// TIA Portal V19 export
FUNCTION_BLOCK "A0302_PareggiatoreTesta_FB"   // FB86, LAD
// stored: MemoryReserve 100, SetENOAutomatically false
   VAR_INPUT
      AreaInterface : "AreaInterface";
      ZSI : "udt_ZoneSafetyInterface";
      DSI_Feed : "udt_DeviceSafetyInterface";
      DSI_Valve : "udt_DeviceSafetyInterface";
      Drive : "TAx_DriveInterface";
      DataIn : Struct
         OP_MoveToPos : Bool;
         Sollevamento : Struct
            OP : "OP_PB";
         END_STRUCT;
         Centraggio : Struct
            OP : "OP_PB";
            AnalSens : Int;
         END_STRUCT;
         Sens { ExternalWritable := 'False'} : Struct
            FTC1_Rall : Bool;   // 2010BF2 - I50.3
            FTC2_Prox_Ls : Bool;   // 2010BF3 - I50.4
            PresenzaMat : Bool;   // FC presenza materiale agganciato lato paregg testa
            FC_Aticoll_Spalla : Bool;
         END_STRUCT;
      END_STRUCT;
      CIn : Struct
         Manager : Struct
            EnableStopDoorOpeningReq { ExternalAccessible := 'False'; ExternalVisible := 'False'; ExternalWritable := 'False'} : Bool;
            EnableStopInPhase { ExternalAccessible := 'False'; ExternalVisible := 'False'; ExternalWritable := 'False'} : Bool;
            EnableStopProgrammed { ExternalAccessible := 'False'; ExternalVisible := 'False'; ExternalWritable := 'False'} : Bool;
            Control_ON { ExternalAccessible := 'False'; ExternalVisible := 'False'; ExternalWritable := 'False'} : Bool;
            MoveToPos { ExternalAccessible := 'False'; ExternalVisible := 'False'; ExternalWritable := 'False'} : Bool;
            Pos { ExternalAccessible := 'False'; ExternalVisible := 'False'; ExternalWritable := 'False'} : LReal;
            Speed : LReal;
            Bloccaggio { ExternalAccessible := 'False'; ExternalVisible := 'False'; ExternalWritable := 'False'} : Struct
               Rest : Bool;
               Work : Bool;
            END_STRUCT;
            Sollevatore { ExternalAccessible := 'False'; ExternalVisible := 'False'; ExternalWritable := 'False'} : Struct
               Rest : Bool;
               Work : Bool;
            END_STRUCT;
            Centraggio { ExternalAccessible := 'False'; ExternalVisible := 'False'; ExternalWritable := 'False'} : Struct
               Rest : Bool;
               Work : Bool;
            END_STRUCT;
         END_STRUCT;
         SemiAut_Pb { ExternalWritable := 'False'} : Bool;
         Bordatrice : Struct
            Ax : "Positioning_EPOS_Machine_COut";
            Sts : Struct
               PosTargetEnable : Bool;
               PosTarget_Reached : Bool;
               In_W_Pos : Bool;
               AtRest : Bool;
            END_STRUCT;
            RegSpalla : Struct
               Infeed_ReqON : Bool;
            END_STRUCT;
         END_STRUCT;
         Rulliera { ExternalWritable := 'False'} : Struct
            Ax_1 : "SpeedMachine_COut";
            Ax_2 : "SpeedMachine_COut";
            Centratori : "ValveMachine_COut";
            Coda : Struct
               Sens : Struct
                  FTC_Rall : Bool;   // Sensori presenza materiale banco rallentamento ingresso
                  FTC_Prox_Ing : Bool;   // Sensori presenza materiale banco limite ingresso
               END_STRUCT;
            END_STRUCT;
            Centro : Struct
               Sens : Struct
                  FTC_Centrale : Bool;   // 2010BF1 - I50.2
               END_STRUCT;
            END_STRUCT;
         END_STRUCT;
         CarroPareggCoda { ExternalWritable := 'False'} : Struct
            Sens : Struct
               FTC_Ingombro_In : Bool;   // 2012BF1 - I50.0
               FTC_Ingombro_Out : Bool;   // 2012BF2 - I50.1
               PresenzaMat : Bool;   // FC presenza materiale agganciato lato paregg coda
            END_STRUCT;
            OilInTargetPressure : Bool;
         END_STRUCT;
         CarriPareggiatori : Struct
            ZoneA0302Entry_Empty { ExternalWritable := 'False'} : Bool;
            ZoneA0302Exit_Empty { ExternalWritable := 'False'} : Bool;
            RequestNewPosition : Bool;
         END_STRUCT;
         Spalle : Struct
            Coda : Struct
               ActualPos : LReal;
            END_STRUCT;
            Testa : Struct
               ActualPos : LReal;
            END_STRUCT;
         END_STRUCT;
         Manipolatore : Struct
            Sollevatore : "ValveMachine_COut";
         END_STRUCT;
         Centratori : Struct
            Sollevamento : "ValveMachine_COut";
         END_STRUCT;
      END_STRUCT;
      Config : Struct
         Ax : "Positioning_DOL_Machine_Config";
         Bloccaggio : "ValveMachine_Config";
         Sollevamento : "ValveMachine_Config";
         Centraggio : "ValveMachine_Config";
         MinDistanzaConSpalla : LReal;
         DelayMissingCondition : Time;
      END_STRUCT;
      HWID : Struct
         Ax_TEL1 : HW_SUBMODULE;
         Enc_IO : HW_SUBMODULE;
      END_STRUCT;
   END_VAR
   VAR_OUTPUT
      MachineInterface : "MachineInterface";
      COut : Struct
         Ax : "Positioning_DOL_Machine_COut";
         Bloccaggio : "ValveMachine_COut";
         Centraggio : "ValveMachine_COut";
         Sollevatore : "ValveMachine_COut";
         Ax_InWPos : Bool;
         Anticipi { ExternalAccessible := 'False'; ExternalVisible := 'False'; ExternalWritable := 'False'} : Struct
            Work : Struct
               Sollevatore : Bool;
               Centraggio : Bool;
            END_STRUCT;
            Rest : Struct
               Sollevatore : Bool;
               Centraggio : Bool;
            END_STRUCT;
         END_STRUCT;
      END_STRUCT;
   END_VAR
   VAR_IN_OUT
      Par : Struct
         Ax : "Positioning_DOL_Machine_Par";
         Ax_Pers : "Positioning_DOL_Machine_Pers_Data";
         Enc : "PosFbk_RTN";
         Ax_Aut : "A0301_Mach_Speed_Par";
         Bloccaggio_Sens : Struct
            "2111B1" : "Analogic_SensorManagement_Par";
            SogliaWork : Real;
         END_STRUCT;
         CarroPareggTesta : Struct
            Delay_StartMove : Time;
            Preset : LReal;
         END_STRUCT;
         Cremaliera : Struct
            Modulo : LReal;
            Passo : LReal;
         END_STRUCT;
      END_STRUCT;
      IEC_SP : Struct
         FTC_Rall : Struct
            TON_PT : Time;
            TOF_PT : Time;
         END_STRUCT;
         FTC_ProxLs : Struct
            TON_PT : Time;
            TOF_PT : Time;
         END_STRUCT;
         FTC_PresentMat : Struct
            TON_PT : Time;
            TOF_PT : Time;
         END_STRUCT;
         Check_2111B1 : Struct
            TON_PT : Time;
         END_STRUCT;
      END_STRUCT;
   END_VAR
   VAR
      Alarm : Struct
         Ax : "Positioning_DOL_Machine_Alr";
         Enc : "PosFbk_Encoder_Alr";
         Bloccaggio : "ValveAlr";
         Centraggio { S7_SetPoint := 'True'} : "ValveAlr";
         Sollevamento { S7_SetPoint := 'True'} : "ValveAlr";
         SensFC_Aticoll_Spalla : Bool;
         Bloccaggio_AnalSens_Issue : Bool;   // Errore soglia lettura pressione su bloccaggio cremaliera
      END_STRUCT;
      Warning : Struct
         Ax : "Positioning_DOL_Machine_Wng";
         Bloccaggio : "ValveMachine_Wng";
         Centraggio { S7_SetPoint := 'True'} : "ValveMachine_Wng";
         Sollevamento { S7_SetPoint := 'True'} : "ValveMachine_Wng";
         MissingCnd : Struct
            OP_REST_Sollevamento : Bool;   // Mancanza comando arresto
            OP_WORK_Sollevamento : Bool;   // Mancanza consenso lavoro
            OP_REST_Centraggio : Bool;   // Mancanza comando arresto
            OP_WORK_Centraggio : Bool;   // Mancanza consenso lavoro
            OP_REST_Bloccaggio : Bool;   // Mancanza comando arresto
            OP_WORK_Bloccaggio : Bool;   // Mancanza consenso lavoro
         END_STRUCT;
         SW_Limit_AntiCollision : Bool;
      END_STRUCT;
      HMI : Struct
         Ax : Struct
            PbPreset : Bool;
            B_Preset_UM2 : Bool;
            PresetValue : LReal;
         END_STRUCT;
      END_STRUCT;
      Sts : Struct
         ReadyForMove : Bool;   // Pronto al movimento
         OP_PTesta_CanMoveFreely : Bool;
         OP_Ax_CanMoveFreely : Bool;
         Op_MoveToPos_Cnd : Bool;
         Sollevamento : Struct
            OP_Rest_Cnd : Bool;
            Op_Work_Cnd : Bool;
         END_STRUCT;
         Centraggio : Struct
            OP_Rest_Cnd : Bool;
            Op_Work_Cnd : Bool;
         END_STRUCT;
      END_STRUCT;
      Ctrl : Struct
         Sollevamento : Struct
            OP_Rest_Man : Bool;
            OP_Work_Man : Bool;
            OP_Rest_Aut : Bool;
            OP_Work_Aut : Bool;
            OP_Rest : Bool;
            OP_Work : Bool;
         END_STRUCT;
         Centraggio : Struct
            OP_Rest_Aut : Bool;
            OP_Work_Aut : Bool;
            OP_Rest_Man : Bool;
            OP_Work_Man : Bool;
            OP_Rest : Bool;
            OP_Work : Bool;
         END_STRUCT;
         Ax : Struct
            OP_MoveToPos_Man : Bool;
            OP_MoveToPos_Aut : Bool;
            OP_MoveToPos : Bool;
         END_STRUCT;
      END_STRUCT;
      AUX : Struct
         OP_MoveToPos : Bool;
         Sollevamento : Struct
            OP_Rest : Bool;
            OP_Work : Bool;
         END_STRUCT;
         Centraggio : Struct
            OP_Rest : Bool;
            OP_Work : Bool;
         END_STRUCT;
      END_STRUCT;
      Ax : "Positioning_DOL_Machine_FB";
      Enc : "PosFbk_SickAFM60";
      Enc_ITF : "PosFbk_ITF";
      Bloccaggio : "ValveMachine_FB";
      Centraggio : "ValveMachine_FB";
      Sollevamento { S7_SetPoint := 'True'} : "ValveMachine_FB";
      TON_Centraggio : Struct
         OP_REST_MissingCnd { S7_SetPoint := 'True'} : TON_TIME;
         OP_WORK_MissingCnd { S7_SetPoint := 'True'} : TON_TIME;
      END_STRUCT;
      TON_Sollevamento : Struct
         OP_REST_MissingCnd { S7_SetPoint := 'True'} : TON_TIME;
         OP_WORK_MissingCnd { S7_SetPoint := 'True'} : TON_TIME;
      END_STRUCT;
      TON_Bloccaggio : Struct
         OP_REST_MissingCnd { S7_SetPoint := 'True'} : TON_TIME;
         OP_WORK_MissingCnd { S7_SetPoint := 'True'} : TON_TIME;
      END_STRUCT;
      IEC_FTC_Rall : Struct
         TON_Delay : IEC_TIMER;
         TOF_Delay { S7_SetPoint := 'True'} : IEC_TIMER;
         FTC_On { S7_SetPoint := 'True'} : Bool;
      END_STRUCT;
      IEC_FTC_ProxLs : Struct
         TON_Delay : IEC_TIMER;
         TOF_Delay { S7_SetPoint := 'True'} : IEC_TIMER;
         FTC_On { S7_SetPoint := 'True'} : Bool;
      END_STRUCT;
      IEC_FTC_PresentMat : Struct
         TON_Delay : IEC_TIMER;
         TOF_Delay { S7_SetPoint := 'True'} : IEC_TIMER;
         FTC_On { S7_SetPoint := 'True'} : Bool;
      END_STRUCT;
      IEC_DelayCheck_2111B1 : IEC_TIMER;
      Bloccaggio_AnalSens { S7_SetPoint := 'True'} : "AnalogThreshold";
      CarroTesta : Struct
         RimanenzaPos : LReal;
         PassoReq : LReal;
         PosBattutePz : LReal;
         SemiBeamLen : LReal;
         NrPassiReq : LReal;
         Pos { ExternalAccessible := 'False'; ExternalVisible := 'False'; ExternalWritable := 'False'} : LReal;   // Posizione calcolata in funzione della cremaliera
      END_STRUCT;
      TON_DistanzaOK : IEC_TIMER;
      TON_Anticipi : Struct
         Rest : Struct
            Sollevamento { S7_SetPoint := 'True'} : IEC_TIMER;
            Centraggio : IEC_TIMER;
         END_STRUCT;
         Work : Struct
            Sollevamento : IEC_TIMER;
            Centraggio { S7_SetPoint := 'True'} : IEC_TIMER;
         END_STRUCT;
      END_STRUCT;
   END_VAR
   VAR_TEMP
      PE : Struct
         OP_MoveToPos : Bool;
         Sollevamento : Struct
            OP_Rest : Bool;
            OP_Work : Bool;
         END_STRUCT;
         Centraggio : Struct
            OP_Rest : Bool;
            OP_Work : Bool;
         END_STRUCT;
      END_STRUCT;
      ActualDifference : LReal;
   END_VAR
   VAR CONSTANT
      RACK_STEP : LReal;   // Passo Cremagliera mm
   END_VAR
   VAR_TEMP   // added for the SCL form of the ladder/FBD networks
      _w1 : Bool;
      _w2 : Bool;
      _w3 : Bool;
      _w4 : Bool;
      _w5 : Bool;
      _w6 : Bool;
      _w7 : Bool;
      _w8 : Bool;
      _w9 : Bool;
      _w10 : Bool;
      _w11 : Bool;
      _w12 : Bool;
   END_VAR
BEGIN

REGION Network 1 (SCL): Reset allarmi
   IF #AreaInterface.RstAlarms THEN
       #Alarm.SensFC_Aticoll_Spalla := FALSE;
       #Alarm.Bloccaggio_AnalSens_Issue := FALSE;
   END_IF;
END_REGION

REGION Network 2: <+>
END_REGION

REGION Network 3: Anticipi Movimento LAVORO
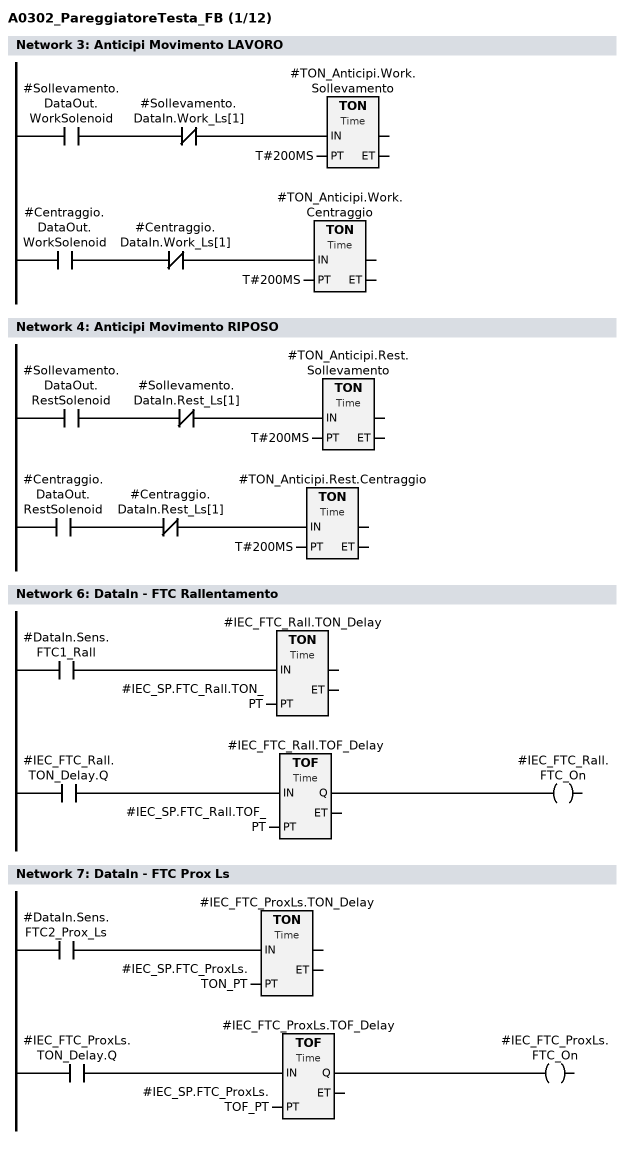
   RUNG wire#powerrail
      Contact( #Sollevamento.DataOut.WorkSolenoid )
      I_Contact( #Sollevamento.DataIn.Work_Ls[1] )
      { S7_Templates := "time_type := Time" } #TON_Anticipi.Work.Sollevamento.TON(pt := T#200MS, et =>)
   END_RUNG
   RUNG wire#powerrail
      Contact( #Centraggio.DataOut.WorkSolenoid )
      I_Contact( #Centraggio.DataIn.Work_Ls[1] )
      { S7_Templates := "time_type := Time" } #TON_Anticipi.Work.Centraggio.TON(pt := T#200MS, et =>)
   END_RUNG
   // the same network as SCL:
   #TON_Anticipi.Work.Sollevamento.TON(IN := #Sollevamento.DataOut.WorkSolenoid AND NOT #Sollevamento.DataIn.Work_Ls[1],
                           PT := T#200MS);
   #TON_Anticipi.Work.Centraggio.TON(IN := #Centraggio.DataOut.WorkSolenoid AND NOT #Centraggio.DataIn.Work_Ls[1],
                           PT := T#200MS);
END_REGION

REGION Network 4: Anticipi Movimento RIPOSO
   RUNG wire#powerrail
      Contact( #Sollevamento.DataOut.RestSolenoid )
      I_Contact( #Sollevamento.DataIn.Rest_Ls[1] )
      { S7_Templates := "time_type := Time" } #TON_Anticipi.Rest.Sollevamento.TON(pt := T#200MS, et =>)
   END_RUNG
   RUNG wire#powerrail
      Contact( #Centraggio.DataOut.RestSolenoid )
      I_Contact( #Centraggio.DataIn.Rest_Ls[1] )
      { S7_Templates := "time_type := Time" } #TON_Anticipi.Rest.Centraggio.TON(pt := T#200MS, et =>)
   END_RUNG
   // the same network as SCL:
   #TON_Anticipi.Rest.Sollevamento.TON(IN := #Sollevamento.DataOut.RestSolenoid AND NOT #Sollevamento.DataIn.Rest_Ls[1],
                           PT := T#200MS);
   #TON_Anticipi.Rest.Centraggio.TON(IN := #Centraggio.DataOut.RestSolenoid AND NOT #Centraggio.DataIn.Rest_Ls[1],
                           PT := T#200MS);
END_REGION

REGION Network 5: <+>
END_REGION

REGION Network 6: DataIn - FTC Rallentamento
   RUNG wire#powerrail
      Contact( #DataIn.Sens.FTC1_Rall )
      { S7_Templates := "time_type := Time" } #IEC_FTC_Rall.TON_Delay.TON(pt := #IEC_SP.FTC_Rall.TON_PT, et =>)
   END_RUNG
   RUNG wire#powerrail
      Contact( #IEC_FTC_Rall.TON_Delay.Q )
      { S7_Templates := "time_type := Time" } #IEC_FTC_Rall.TOF_Delay.TOF(pt := #IEC_SP.FTC_Rall.TOF_PT, et =>)
      Coil( #IEC_FTC_Rall.FTC_On )
   END_RUNG
   // the same network as SCL:
   #IEC_FTC_Rall.TON_Delay.TON(IN := #DataIn.Sens.FTC1_Rall, PT := #IEC_SP.FTC_Rall.TON_PT);
   #IEC_FTC_Rall.TOF_Delay.TOF(IN := #IEC_FTC_Rall.TON_Delay.Q, PT := #IEC_SP.FTC_Rall.TOF_PT);
   #IEC_FTC_Rall.FTC_On := #IEC_FTC_Rall.TOF_Delay.Q;
END_REGION

REGION Network 7: DataIn - FTC Prox Ls
   RUNG wire#powerrail
      Contact( #DataIn.Sens.FTC2_Prox_Ls )
      { S7_Templates := "time_type := Time" } #IEC_FTC_ProxLs.TON_Delay.TON(pt := #IEC_SP.FTC_ProxLs.TON_PT, et =>)
   END_RUNG
   RUNG wire#powerrail
      Contact( #IEC_FTC_ProxLs.TON_Delay.Q )
      { S7_Templates := "time_type := Time" } #IEC_FTC_ProxLs.TOF_Delay.TOF(pt := #IEC_SP.FTC_ProxLs.TOF_PT, et =>)
      Coil( #IEC_FTC_ProxLs.FTC_On )
   END_RUNG
   // the same network as SCL:
   #IEC_FTC_ProxLs.TON_Delay.TON(IN := #DataIn.Sens.FTC2_Prox_Ls, PT := #IEC_SP.FTC_ProxLs.TON_PT);
   #IEC_FTC_ProxLs.TOF_Delay.TOF(IN := #IEC_FTC_ProxLs.TON_Delay.Q, PT := #IEC_SP.FTC_ProxLs.TOF_PT);
   #IEC_FTC_ProxLs.FTC_On := #IEC_FTC_ProxLs.TOF_Delay.Q;
END_REGION

REGION Network 8: DataIn - FTC Presenza materiale
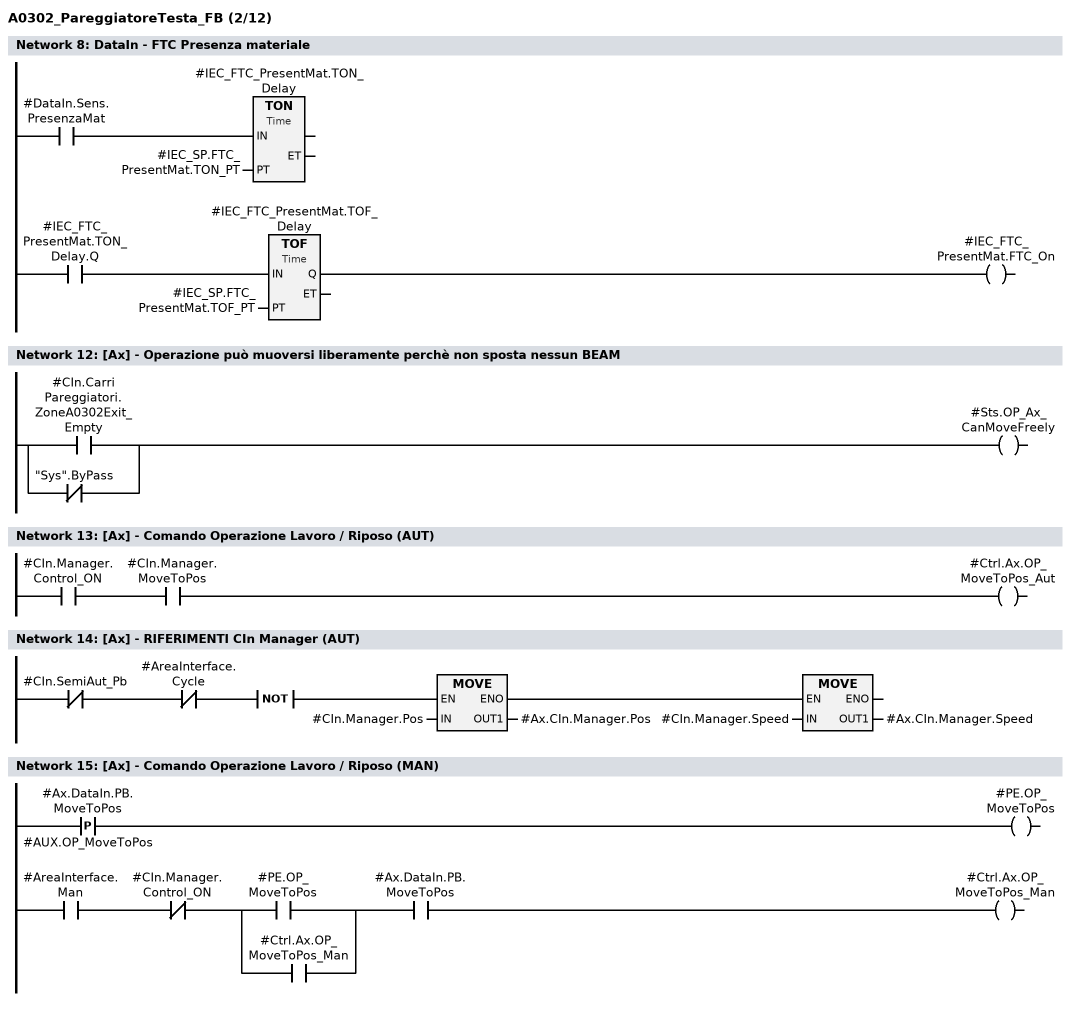
   RUNG wire#powerrail
      Contact( #DataIn.Sens.PresenzaMat )
      { S7_Templates := "time_type := Time" } #IEC_FTC_PresentMat.TON_Delay.TON(pt := #IEC_SP.FTC_PresentMat.TON_PT, et =>)
   END_RUNG
   RUNG wire#powerrail
      Contact( #IEC_FTC_PresentMat.TON_Delay.Q )
      { S7_Templates := "time_type := Time" } #IEC_FTC_PresentMat.TOF_Delay.TOF(pt := #IEC_SP.FTC_PresentMat.TOF_PT, et =>)
      Coil( #IEC_FTC_PresentMat.FTC_On )
   END_RUNG
   // the same network as SCL:
   #IEC_FTC_PresentMat.TON_Delay.TON(IN := #DataIn.Sens.PresenzaMat, PT := #IEC_SP.FTC_PresentMat.TON_PT);
   #IEC_FTC_PresentMat.TOF_Delay.TOF(IN := #IEC_FTC_PresentMat.TON_Delay.Q, PT := #IEC_SP.FTC_PresentMat.TOF_PT);
   #IEC_FTC_PresentMat.FTC_On := #IEC_FTC_PresentMat.TOF_Delay.Q;
END_REGION

REGION Network 9: <+>
END_REGION

REGION Network 10: <<< CARRO PAREGGIATORE TESTA >>>
END_REGION

REGION Network 11: <+>
END_REGION

REGION Network 12: [Ax] - Operazione può muoversi liberamente perchè non sposta nessun BEAM
   RUNG wire#powerrail
      Contact( #CIn.CarriPareggiatori.ZoneA0302Exit_Empty )
      wire#w1
      Coil( #Sts.OP_Ax_CanMoveFreely )
   END_RUNG
   RUNG wire#powerrail
      I_Contact( "Sys".ByPass )
   END_RUNG wire#w1
   // the same network as SCL:
   #Sts.OP_Ax_CanMoveFreely := #CIn.CarriPareggiatori.ZoneA0302Exit_Empty OR NOT "Sys".ByPass;
END_REGION

REGION Network 13: [Ax] - Comando Operazione Lavoro / Riposo (AUT)
   RUNG wire#powerrail
      Contact( #CIn.Manager.Control_ON )
      Contact( #CIn.Manager.MoveToPos )
      Coil( #Ctrl.Ax.OP_MoveToPos_Aut )
   END_RUNG
   // the same network as SCL:
   #Ctrl.Ax.OP_MoveToPos_Aut := #CIn.Manager.Control_ON AND #CIn.Manager.MoveToPos;
END_REGION

REGION Network 14: [Ax] - RIFERIMENTI CIn Manager (AUT)
   RUNG wire#powerrail
      I_Contact( #CIn.SemiAut_Pb )
      I_Contact( #AreaInterface.Cycle )
      Not()
      Move(in := #CIn.Manager.Pos, out1 => #Ax.CIn.Manager.Pos)
      Move(in := #CIn.Manager.Speed, out1 => #Ax.CIn.Manager.Speed)
   END_RUNG
   // the same network as SCL:
   IF NOT (NOT #CIn.SemiAut_Pb AND NOT #AreaInterface.Cycle) THEN
       #Ax.CIn.Manager.Pos := #CIn.Manager.Pos;
       #Ax.CIn.Manager.Speed := #CIn.Manager.Speed;
   END_IF;
END_REGION

REGION Network 15: [Ax] - Comando Operazione Lavoro / Riposo (MAN)
   RUNG wire#powerrail
      P_Contact(operand := #Ax.DataIn.PB.MoveToPos, bit := #AUX.OP_MoveToPos)
      Coil( #PE.OP_MoveToPos )
   END_RUNG
   RUNG wire#powerrail
      Contact( #AreaInterface.Man )
      I_Contact( #CIn.Manager.Control_ON )
      wire#w1
      Contact( #PE.OP_MoveToPos )
      wire#w2
      Contact( #Ax.DataIn.PB.MoveToPos )
      Coil( #Ctrl.Ax.OP_MoveToPos_Man )
   END_RUNG
   RUNG wire#w1
      Contact( #Ctrl.Ax.OP_MoveToPos_Man )
   END_RUNG wire#w2
   // the same network as SCL:
   #_w1 := #Ax.DataIn.PB.MoveToPos AND NOT #AUX.OP_MoveToPos;   // rising edge of #Ax.DataIn.PB.MoveToPos
   #AUX.OP_MoveToPos := #Ax.DataIn.PB.MoveToPos;
   #PE.OP_MoveToPos := #_w1;
   #Ctrl.Ax.OP_MoveToPos_Man := #AreaInterface.Man AND NOT #CIn.Manager.Control_ON AND (#PE.OP_MoveToPos OR #Ctrl.Ax.OP_MoveToPos_Man) AND #Ax.DataIn.PB.MoveToPos;
END_REGION

REGION Network 16: <+>
END_REGION

REGION Network 17: [Sollevam + Centraggio] - Operazione può muoversi liberamente perchè non sposta nessun BEAM
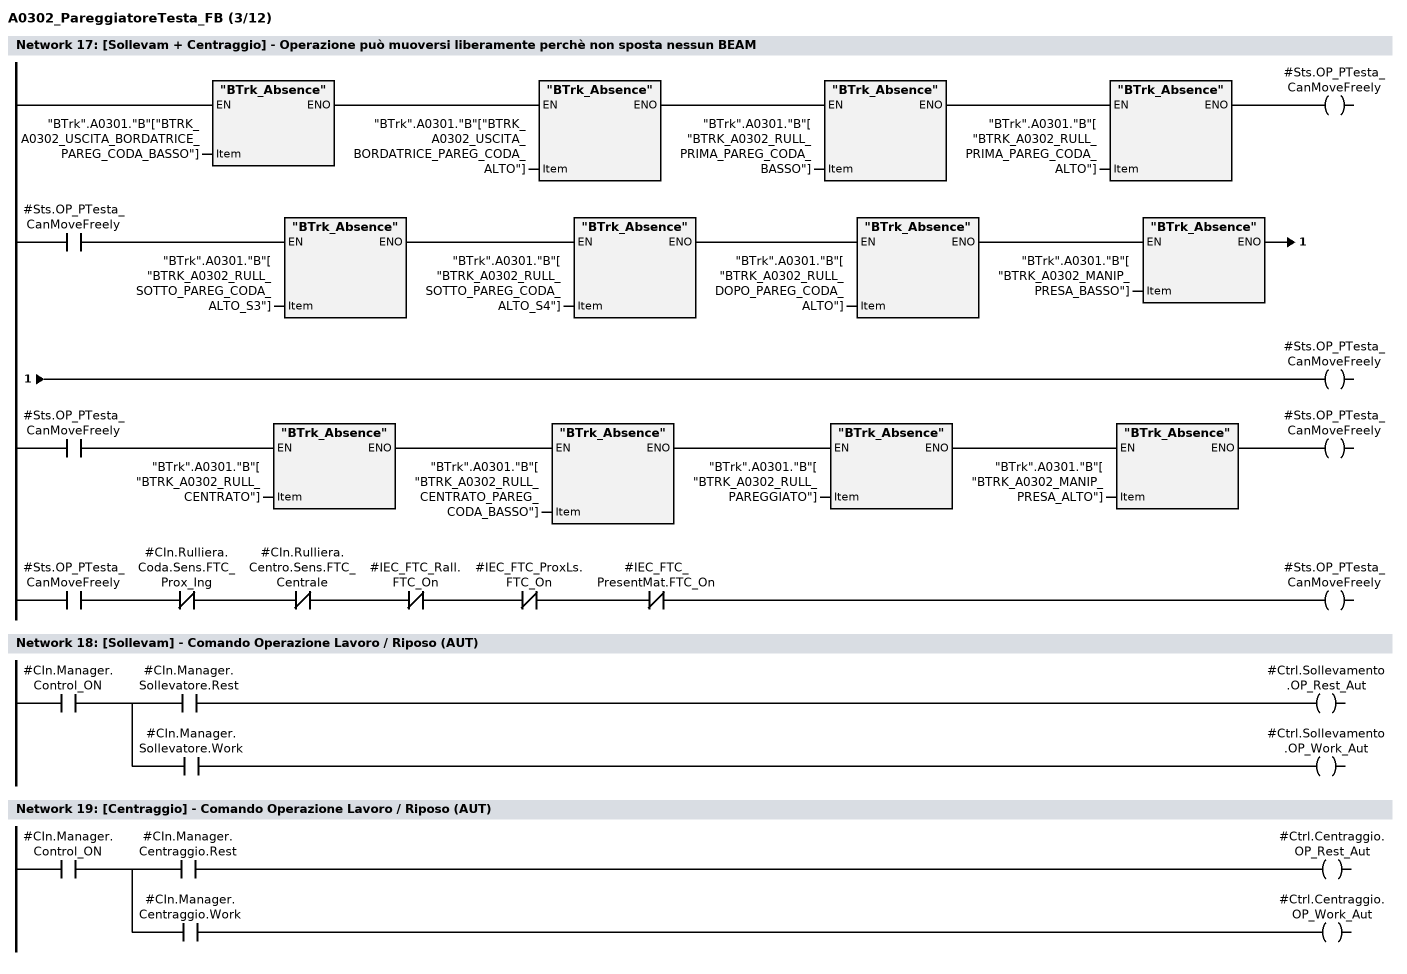
   RUNG wire#powerrail
      "BTrk_Absence"(Item := "BTrk".A0301."B"["BTRK_A0302_USCITA_BORDATRICE_PAREG_CODA_BASSO"])
      "BTrk_Absence"(Item := "BTrk".A0301."B"["BTRK_A0302_USCITA_BORDATRICE_PAREG_CODA_ALTO"])
      "BTrk_Absence"(Item := "BTrk".A0301."B"["BTRK_A0302_RULL_PRIMA_PAREG_CODA_BASSO"])
      "BTrk_Absence"(Item := "BTrk".A0301."B"["BTRK_A0302_RULL_PRIMA_PAREG_CODA_ALTO"])
      Coil( #Sts.OP_PTesta_CanMoveFreely )
   END_RUNG
   RUNG wire#powerrail
      Contact( #Sts.OP_PTesta_CanMoveFreely )
      "BTrk_Absence"(Item := "BTrk".A0301."B"["BTRK_A0302_RULL_SOTTO_PAREG_CODA_ALTO_S3"])
      "BTrk_Absence"(Item := "BTrk".A0301."B"["BTRK_A0302_RULL_SOTTO_PAREG_CODA_ALTO_S4"])
      "BTrk_Absence"(Item := "BTrk".A0301."B"["BTRK_A0302_RULL_DOPO_PAREG_CODA_ALTO"])
      "BTrk_Absence"(Item := "BTrk".A0301."B"["BTRK_A0302_MANIP_PRESA_BASSO"])
      Coil( #Sts.OP_PTesta_CanMoveFreely )
   END_RUNG
   RUNG wire#powerrail
      Contact( #Sts.OP_PTesta_CanMoveFreely )
      "BTrk_Absence"(Item := "BTrk".A0301."B"["BTRK_A0302_RULL_CENTRATO"])
      "BTrk_Absence"(Item := "BTrk".A0301."B"["BTRK_A0302_RULL_CENTRATO_PAREG_CODA_BASSO"])
      "BTrk_Absence"(Item := "BTrk".A0301."B"["BTRK_A0302_RULL_PAREGGIATO"])
      "BTrk_Absence"(Item := "BTrk".A0301."B"["BTRK_A0302_MANIP_PRESA_ALTO"])
      Coil( #Sts.OP_PTesta_CanMoveFreely )
   END_RUNG
   RUNG wire#powerrail
      Contact( #Sts.OP_PTesta_CanMoveFreely )
      I_Contact( #CIn.Rulliera.Coda.Sens.FTC_Prox_Ing )
      I_Contact( #CIn.Rulliera.Centro.Sens.FTC_Centrale )
      I_Contact( #IEC_FTC_Rall.FTC_On )
      I_Contact( #IEC_FTC_ProxLs.FTC_On )
      I_Contact( #IEC_FTC_PresentMat.FTC_On )
      Coil( #Sts.OP_PTesta_CanMoveFreely )
   END_RUNG
   // the same network as SCL:
   "BTrk_Absence"(Item := "BTrk".A0301."B"["BTRK_A0302_USCITA_BORDATRICE_PAREG_CODA_BASSO"], ENO => #_w1);
   "BTrk_Absence"(EN := #_w1,
                  Item := "BTrk".A0301."B"["BTRK_A0302_USCITA_BORDATRICE_PAREG_CODA_ALTO"],
                  ENO => #_w2);
   "BTrk_Absence"(EN := #_w2, Item := "BTrk".A0301."B"["BTRK_A0302_RULL_PRIMA_PAREG_CODA_BASSO"], ENO => #_w3);
   "BTrk_Absence"(EN := #_w3, Item := "BTrk".A0301."B"["BTRK_A0302_RULL_PRIMA_PAREG_CODA_ALTO"], ENO => #_w4);
   #Sts.OP_PTesta_CanMoveFreely := #_w4;
   "BTrk_Absence"(EN := #Sts.OP_PTesta_CanMoveFreely,
                  Item := "BTrk".A0301."B"["BTRK_A0302_RULL_SOTTO_PAREG_CODA_ALTO_S3"],
                  ENO => #_w5);
   "BTrk_Absence"(EN := #_w5, Item := "BTrk".A0301."B"["BTRK_A0302_RULL_SOTTO_PAREG_CODA_ALTO_S4"], ENO => #_w6);
   "BTrk_Absence"(EN := #_w6, Item := "BTrk".A0301."B"["BTRK_A0302_RULL_DOPO_PAREG_CODA_ALTO"], ENO => #_w7);
   "BTrk_Absence"(EN := #_w7, Item := "BTrk".A0301."B"["BTRK_A0302_MANIP_PRESA_BASSO"], ENO => #_w8);
   #Sts.OP_PTesta_CanMoveFreely := #_w8;
   "BTrk_Absence"(EN := #Sts.OP_PTesta_CanMoveFreely,
                  Item := "BTrk".A0301."B"["BTRK_A0302_RULL_CENTRATO"],
                  ENO => #_w9);
   "BTrk_Absence"(EN := #_w9,
                  Item := "BTrk".A0301."B"["BTRK_A0302_RULL_CENTRATO_PAREG_CODA_BASSO"],
                  ENO => #_w10);
   "BTrk_Absence"(EN := #_w10, Item := "BTrk".A0301."B"["BTRK_A0302_RULL_PAREGGIATO"], ENO => #_w11);
   "BTrk_Absence"(EN := #_w11, Item := "BTrk".A0301."B"["BTRK_A0302_MANIP_PRESA_ALTO"], ENO => #_w12);
   #Sts.OP_PTesta_CanMoveFreely := #_w12;
   #Sts.OP_PTesta_CanMoveFreely := #Sts.OP_PTesta_CanMoveFreely AND NOT #CIn.Rulliera.Coda.Sens.FTC_Prox_Ing AND NOT #CIn.Rulliera.Centro.Sens.FTC_Centrale AND NOT #IEC_FTC_Rall.FTC_On AND NOT #IEC_FTC_ProxLs.FTC_On AND NOT #IEC_FTC_PresentMat.FTC_On;
END_REGION

REGION Network 18: [Sollevam] - Comando Operazione Lavoro / Riposo (AUT)
   RUNG wire#powerrail
      Contact( #CIn.Manager.Control_ON )
      wire#w1
      Contact( #CIn.Manager.Sollevatore.Rest )
      Coil( #Ctrl.Sollevamento.OP_Rest_Aut )
   END_RUNG
   RUNG wire#w1
      Contact( #CIn.Manager.Sollevatore.Work )
      Coil( #Ctrl.Sollevamento.OP_Work_Aut )
   END_RUNG
   // the same network as SCL:
   #Ctrl.Sollevamento.OP_Rest_Aut := #CIn.Manager.Control_ON AND #CIn.Manager.Sollevatore.Rest;
   #Ctrl.Sollevamento.OP_Work_Aut := #CIn.Manager.Control_ON AND #CIn.Manager.Sollevatore.Work;
END_REGION

REGION Network 19: [Centraggio] - Comando Operazione Lavoro / Riposo (AUT)
   RUNG wire#powerrail
      Contact( #CIn.Manager.Control_ON )
      wire#w1
      Contact( #CIn.Manager.Centraggio.Rest )
      Coil( #Ctrl.Centraggio.OP_Rest_Aut )
   END_RUNG
   RUNG wire#w1
      Contact( #CIn.Manager.Centraggio.Work )
      Coil( #Ctrl.Centraggio.OP_Work_Aut )
   END_RUNG
   // the same network as SCL:
   #Ctrl.Centraggio.OP_Rest_Aut := #CIn.Manager.Control_ON AND #CIn.Manager.Centraggio.Rest;
   #Ctrl.Centraggio.OP_Work_Aut := #CIn.Manager.Control_ON AND #CIn.Manager.Centraggio.Work;
END_REGION

REGION Network 20: <+>
END_REGION

REGION Network 21: [Sollevam] - Comando Operazione Lavoro / Riposo (MAN)
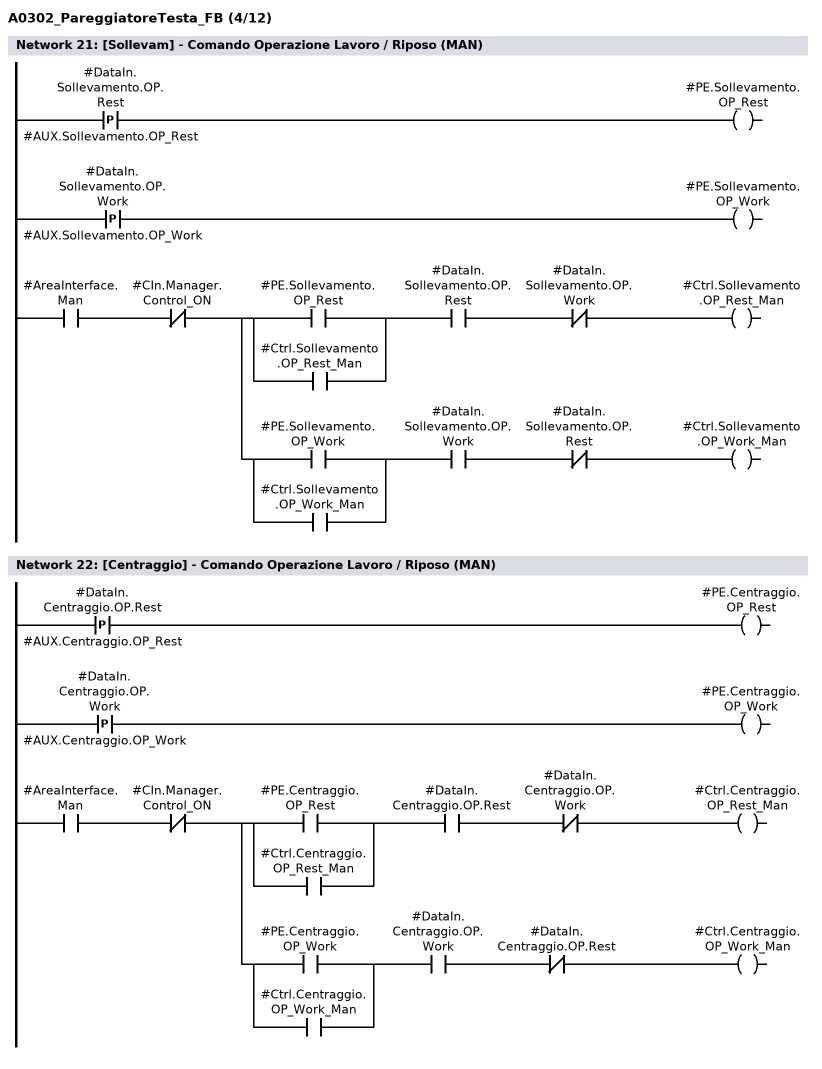
   RUNG wire#powerrail
      P_Contact(operand := #DataIn.Sollevamento.OP.Rest, bit := #AUX.Sollevamento.OP_Rest)
      Coil( #PE.Sollevamento.OP_Rest )
   END_RUNG
   RUNG wire#powerrail
      P_Contact(operand := #DataIn.Sollevamento.OP.Work, bit := #AUX.Sollevamento.OP_Work)
      Coil( #PE.Sollevamento.OP_Work )
   END_RUNG
   RUNG wire#powerrail
      Contact( #AreaInterface.Man )
      I_Contact( #CIn.Manager.Control_ON )
      wire#w1
      Contact( #PE.Sollevamento.OP_Rest )
      wire#w2
      Contact( #DataIn.Sollevamento.OP.Rest )
      I_Contact( #DataIn.Sollevamento.OP.Work )
      Coil( #Ctrl.Sollevamento.OP_Rest_Man )
   END_RUNG
   RUNG wire#w1
      Contact( #Ctrl.Sollevamento.OP_Rest_Man )
   END_RUNG wire#w2
   RUNG wire#w1
      Contact( #PE.Sollevamento.OP_Work )
      wire#w3
      Contact( #DataIn.Sollevamento.OP.Work )
      I_Contact( #DataIn.Sollevamento.OP.Rest )
      Coil( #Ctrl.Sollevamento.OP_Work_Man )
   END_RUNG
   RUNG wire#w1
      Contact( #Ctrl.Sollevamento.OP_Work_Man )
   END_RUNG wire#w3
   // the same network as SCL:
   #_w1 := #DataIn.Sollevamento.OP.Rest AND NOT #AUX.Sollevamento.OP_Rest;   // rising edge of #DataIn.Sollevamento.OP.Rest
   #AUX.Sollevamento.OP_Rest := #DataIn.Sollevamento.OP.Rest;
   #PE.Sollevamento.OP_Rest := #_w1;
   #_w2 := #DataIn.Sollevamento.OP.Work AND NOT #AUX.Sollevamento.OP_Work;   // rising edge of #DataIn.Sollevamento.OP.Work
   #AUX.Sollevamento.OP_Work := #DataIn.Sollevamento.OP.Work;
   #PE.Sollevamento.OP_Work := #_w2;
   #_w3 := #AreaInterface.Man AND NOT #CIn.Manager.Control_ON;
   #Ctrl.Sollevamento.OP_Rest_Man := #_w3 AND (#PE.Sollevamento.OP_Rest OR #Ctrl.Sollevamento.OP_Rest_Man) AND #DataIn.Sollevamento.OP.Rest AND NOT #DataIn.Sollevamento.OP.Work;
   #Ctrl.Sollevamento.OP_Work_Man := #_w3 AND (#PE.Sollevamento.OP_Work OR #Ctrl.Sollevamento.OP_Work_Man) AND #DataIn.Sollevamento.OP.Work AND NOT #DataIn.Sollevamento.OP.Rest;
END_REGION

REGION Network 22: [Centraggio] - Comando Operazione Lavoro / Riposo (MAN)
   RUNG wire#powerrail
      P_Contact(operand := #DataIn.Centraggio.OP.Rest, bit := #AUX.Centraggio.OP_Rest)
      Coil( #PE.Centraggio.OP_Rest )
   END_RUNG
   RUNG wire#powerrail
      P_Contact(operand := #DataIn.Centraggio.OP.Work, bit := #AUX.Centraggio.OP_Work)
      Coil( #PE.Centraggio.OP_Work )
   END_RUNG
   RUNG wire#powerrail
      Contact( #AreaInterface.Man )
      I_Contact( #CIn.Manager.Control_ON )
      wire#w1
      Contact( #PE.Centraggio.OP_Rest )
      wire#w2
      Contact( #DataIn.Centraggio.OP.Rest )
      I_Contact( #DataIn.Centraggio.OP.Work )
      Coil( #Ctrl.Centraggio.OP_Rest_Man )
   END_RUNG
   RUNG wire#w1
      Contact( #Ctrl.Centraggio.OP_Rest_Man )
   END_RUNG wire#w2
   RUNG wire#w1
      Contact( #PE.Centraggio.OP_Work )
      wire#w3
      Contact( #DataIn.Centraggio.OP.Work )
      I_Contact( #DataIn.Centraggio.OP.Rest )
      Coil( #Ctrl.Centraggio.OP_Work_Man )
   END_RUNG
   RUNG wire#w1
      Contact( #Ctrl.Centraggio.OP_Work_Man )
   END_RUNG wire#w3
   // the same network as SCL:
   #_w1 := #DataIn.Centraggio.OP.Rest AND NOT #AUX.Centraggio.OP_Rest;   // rising edge of #DataIn.Centraggio.OP.Rest
   #AUX.Centraggio.OP_Rest := #DataIn.Centraggio.OP.Rest;
   #PE.Centraggio.OP_Rest := #_w1;
   #_w2 := #DataIn.Centraggio.OP.Work AND NOT #AUX.Centraggio.OP_Work;   // rising edge of #DataIn.Centraggio.OP.Work
   #AUX.Centraggio.OP_Work := #DataIn.Centraggio.OP.Work;
   #PE.Centraggio.OP_Work := #_w2;
   #_w3 := #AreaInterface.Man AND NOT #CIn.Manager.Control_ON;
   #Ctrl.Centraggio.OP_Rest_Man := #_w3 AND (#PE.Centraggio.OP_Rest OR #Ctrl.Centraggio.OP_Rest_Man) AND #DataIn.Centraggio.OP.Rest AND NOT #DataIn.Centraggio.OP.Work;
   #Ctrl.Centraggio.OP_Work_Man := #_w3 AND (#PE.Centraggio.OP_Work OR #Ctrl.Centraggio.OP_Work_Man) AND #DataIn.Centraggio.OP.Work AND NOT #DataIn.Centraggio.OP.Rest;
END_REGION

REGION Network 23: <+>
END_REGION

REGION Network 24: Carro Pareggiatore di Testa - Cumulativo Operazione Lavoro / Riposo (ALL)
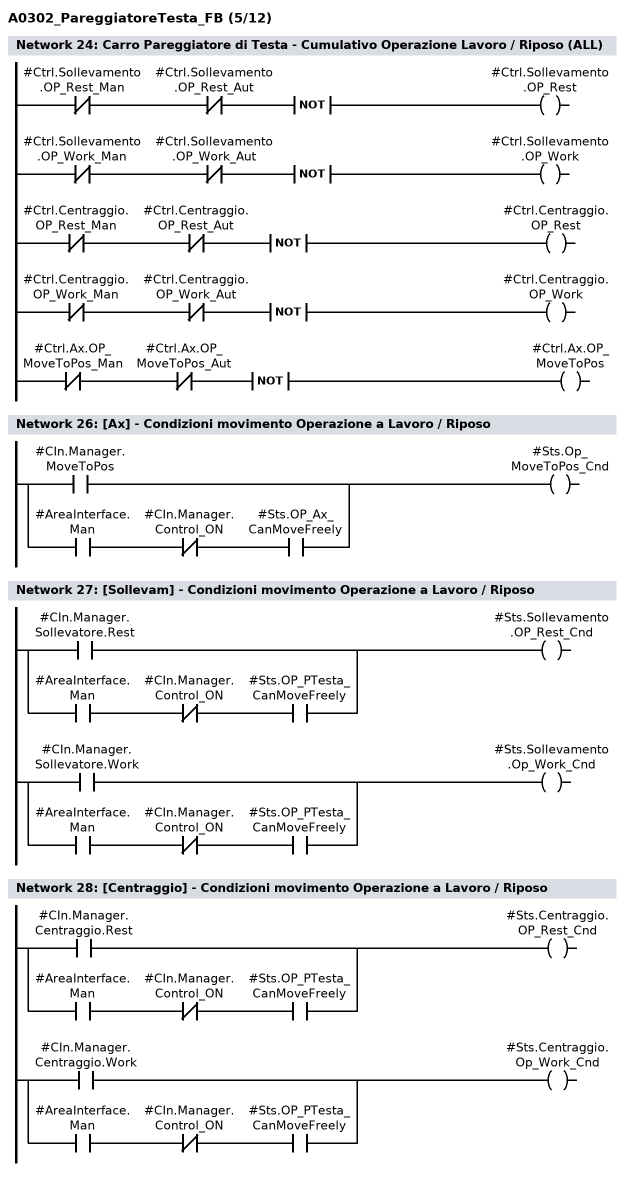
   RUNG wire#powerrail
      I_Contact( #Ctrl.Sollevamento.OP_Rest_Man )
      I_Contact( #Ctrl.Sollevamento.OP_Rest_Aut )
      Not()
      Coil( #Ctrl.Sollevamento.OP_Rest )
   END_RUNG
   RUNG wire#powerrail
      I_Contact( #Ctrl.Sollevamento.OP_Work_Man )
      I_Contact( #Ctrl.Sollevamento.OP_Work_Aut )
      Not()
      Coil( #Ctrl.Sollevamento.OP_Work )
   END_RUNG
   RUNG wire#powerrail
      I_Contact( #Ctrl.Centraggio.OP_Rest_Man )
      I_Contact( #Ctrl.Centraggio.OP_Rest_Aut )
      Not()
      Coil( #Ctrl.Centraggio.OP_Rest )
   END_RUNG
   RUNG wire#powerrail
      I_Contact( #Ctrl.Centraggio.OP_Work_Man )
      I_Contact( #Ctrl.Centraggio.OP_Work_Aut )
      Not()
      Coil( #Ctrl.Centraggio.OP_Work )
   END_RUNG
   RUNG wire#powerrail
      I_Contact( #Ctrl.Ax.OP_MoveToPos_Man )
      I_Contact( #Ctrl.Ax.OP_MoveToPos_Aut )
      Not()
      Coil( #Ctrl.Ax.OP_MoveToPos )
   END_RUNG
   // the same network as SCL:
   #Ctrl.Sollevamento.OP_Rest := NOT (NOT #Ctrl.Sollevamento.OP_Rest_Man AND NOT #Ctrl.Sollevamento.OP_Rest_Aut);
   #Ctrl.Sollevamento.OP_Work := NOT (NOT #Ctrl.Sollevamento.OP_Work_Man AND NOT #Ctrl.Sollevamento.OP_Work_Aut);
   #Ctrl.Centraggio.OP_Rest := NOT (NOT #Ctrl.Centraggio.OP_Rest_Man AND NOT #Ctrl.Centraggio.OP_Rest_Aut);
   #Ctrl.Centraggio.OP_Work := NOT (NOT #Ctrl.Centraggio.OP_Work_Man AND NOT #Ctrl.Centraggio.OP_Work_Aut);
   #Ctrl.Ax.OP_MoveToPos := NOT (NOT #Ctrl.Ax.OP_MoveToPos_Man AND NOT #Ctrl.Ax.OP_MoveToPos_Aut);
END_REGION

REGION Network 25: <+>
END_REGION

REGION Network 26: [Ax] - Condizioni movimento Operazione a Lavoro / Riposo
   RUNG wire#powerrail
      Contact( #CIn.Manager.MoveToPos )
      wire#w1
      Coil( #Sts.Op_MoveToPos_Cnd )
   END_RUNG
   RUNG wire#powerrail
      Contact( #AreaInterface.Man )
      I_Contact( #CIn.Manager.Control_ON )
      Contact( #Sts.OP_Ax_CanMoveFreely )
   END_RUNG wire#w1
   // the same network as SCL:
   #Sts.Op_MoveToPos_Cnd := #CIn.Manager.MoveToPos OR (#AreaInterface.Man AND NOT #CIn.Manager.Control_ON AND #Sts.OP_Ax_CanMoveFreely);
END_REGION

REGION Network 27: [Sollevam] - Condizioni movimento Operazione a Lavoro / Riposo
   RUNG wire#powerrail
      Contact( #CIn.Manager.Sollevatore.Rest )
      wire#w1
      Coil( #Sts.Sollevamento.OP_Rest_Cnd )
   END_RUNG
   RUNG wire#powerrail
      Contact( #AreaInterface.Man )
      I_Contact( #CIn.Manager.Control_ON )
      Contact( #Sts.OP_PTesta_CanMoveFreely )
   END_RUNG wire#w1
   RUNG wire#powerrail
      Contact( #CIn.Manager.Sollevatore.Work )
      wire#w2
      Coil( #Sts.Sollevamento.Op_Work_Cnd )
   END_RUNG
   RUNG wire#powerrail
      Contact( #AreaInterface.Man )
      I_Contact( #CIn.Manager.Control_ON )
      Contact( #Sts.OP_PTesta_CanMoveFreely )
   END_RUNG wire#w2
   // the same network as SCL:
   #Sts.Sollevamento.OP_Rest_Cnd := #CIn.Manager.Sollevatore.Rest OR (#AreaInterface.Man AND NOT #CIn.Manager.Control_ON AND #Sts.OP_PTesta_CanMoveFreely);
   #Sts.Sollevamento.Op_Work_Cnd := #CIn.Manager.Sollevatore.Work OR (#AreaInterface.Man AND NOT #CIn.Manager.Control_ON AND #Sts.OP_PTesta_CanMoveFreely);
END_REGION

REGION Network 28: [Centraggio] - Condizioni movimento Operazione a Lavoro / Riposo
   RUNG wire#powerrail
      Contact( #CIn.Manager.Centraggio.Rest )
      wire#w1
      Coil( #Sts.Centraggio.OP_Rest_Cnd )
   END_RUNG
   RUNG wire#powerrail
      Contact( #AreaInterface.Man )
      I_Contact( #CIn.Manager.Control_ON )
      Contact( #Sts.OP_PTesta_CanMoveFreely )
   END_RUNG wire#w1
   RUNG wire#powerrail
      Contact( #CIn.Manager.Centraggio.Work )
      wire#w2
      Coil( #Sts.Centraggio.Op_Work_Cnd )
   END_RUNG
   RUNG wire#powerrail
      Contact( #AreaInterface.Man )
      I_Contact( #CIn.Manager.Control_ON )
      Contact( #Sts.OP_PTesta_CanMoveFreely )
   END_RUNG wire#w2
   // the same network as SCL:
   #Sts.Centraggio.OP_Rest_Cnd := #CIn.Manager.Centraggio.Rest OR (#AreaInterface.Man AND NOT #CIn.Manager.Control_ON AND #Sts.OP_PTesta_CanMoveFreely);
   #Sts.Centraggio.Op_Work_Cnd := #CIn.Manager.Centraggio.Work OR (#AreaInterface.Man AND NOT #CIn.Manager.Control_ON AND #Sts.OP_PTesta_CanMoveFreely);
END_REGION

REGION Network 29: <+>
END_REGION

REGION Network 30 (SCL): Carro Pareggiatore di Testa - CIn Abilitazioni Stop Manager
   #Sollevamento.Cin.Manager.EnableStopDoorOpeningReq := #Centraggio.Cin.Manager.EnableStopDoorOpeningReq
   := #Bloccaggio.Cin.Manager.EnableStopDoorOpeningReq := #Ax.CIn.Manager.EnableStopDoorOpeningReq := #CIn.Manager.EnableStopDoorOpeningReq;

   #Sollevamento.Cin.Manager.EnableStopInPhase := #Centraggio.Cin.Manager.EnableStopInPhase
   := #Bloccaggio.Cin.Manager.EnableStopInPhase := #Ax.CIn.Manager.EnableStopInPhase := #CIn.Manager.EnableStopInPhase;

   #Sollevamento.Cin.Manager.EnableStopProgrammed := #Centraggio.Cin.Manager.EnableStopProgrammed
   := #Bloccaggio.Cin.Manager.EnableStopProgrammed := #Ax.CIn.Manager.EnableStopProgrammed := #CIn.Manager.EnableStopProgrammed;
END_REGION

REGION Network 31: <+>
END_REGION

REGION Network 32: <<< BLOCCAGGIO SU CREMAGLIERA >>>
END_REGION

REGION Network 33: [Bloccaggio] - Cin Manager (Esecuzione sequenza comandi)
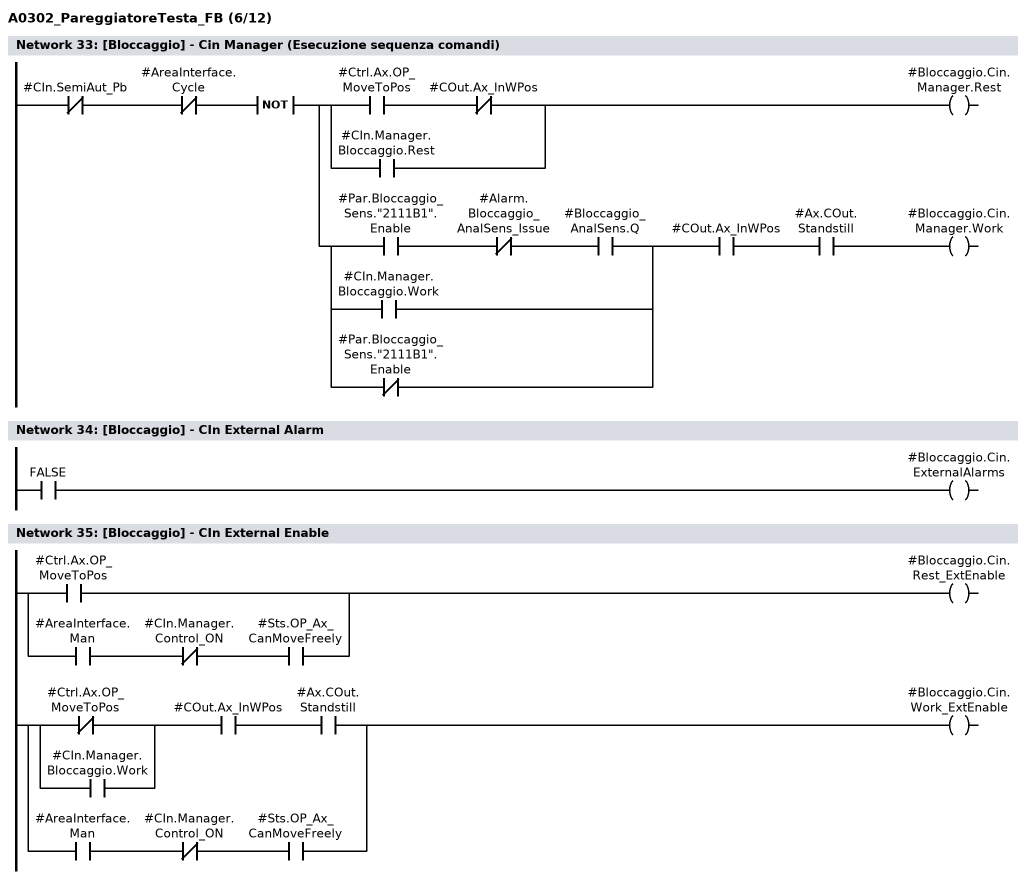
   RUNG wire#powerrail
      I_Contact( #CIn.SemiAut_Pb )
      I_Contact( #AreaInterface.Cycle )
      Not()
      wire#w1
      Contact( #Ctrl.Ax.OP_MoveToPos )
      I_Contact( #COut.Ax_InWPos )
      wire#w2
      Coil( #Bloccaggio.Cin.Manager.Rest )
   END_RUNG
   RUNG wire#w1
      Contact( #CIn.Manager.Bloccaggio.Rest )
   END_RUNG wire#w2
   RUNG wire#w1
      Contact( #Par.Bloccaggio_Sens."2111B1".Enable )
      I_Contact( #Alarm.Bloccaggio_AnalSens_Issue )
      Contact( #Bloccaggio_AnalSens.Q )
      wire#w3
      Contact( #COut.Ax_InWPos )
      Contact( #Ax.COut.Standstill )
      Coil( #Bloccaggio.Cin.Manager.Work )
   END_RUNG
   RUNG wire#w1
      Contact( #CIn.Manager.Bloccaggio.Work )
   END_RUNG wire#w3
   RUNG wire#w1
      I_Contact( #Par.Bloccaggio_Sens."2111B1".Enable )
   END_RUNG wire#w3
   // the same network as SCL:
   #_w1 := NOT (NOT #CIn.SemiAut_Pb AND NOT #AreaInterface.Cycle);
   #Bloccaggio.Cin.Manager.Rest := #_w1 AND ((#Ctrl.Ax.OP_MoveToPos AND NOT #COut.Ax_InWPos) OR #CIn.Manager.Bloccaggio.Rest);
   #Bloccaggio.Cin.Manager.Work := #_w1 AND ((#Par.Bloccaggio_Sens."2111B1".Enable AND NOT #Alarm.Bloccaggio_AnalSens_Issue AND #Bloccaggio_AnalSens.Q) OR #CIn.Manager.Bloccaggio.Work OR NOT #Par.Bloccaggio_Sens."2111B1".Enable) AND #COut.Ax_InWPos AND #Ax.COut.Standstill;
END_REGION

REGION Network 34: [Bloccaggio] - CIn External Alarm
   RUNG wire#powerrail
      Contact( FALSE )
      Coil( #Bloccaggio.Cin.ExternalAlarms )
   END_RUNG
   // the same network as SCL:
   #Bloccaggio.Cin.ExternalAlarms := FALSE;
END_REGION

REGION Network 35: [Bloccaggio] - CIn External Enable
   RUNG wire#powerrail
      Contact( #Ctrl.Ax.OP_MoveToPos )
      wire#w1
      Coil( #Bloccaggio.Cin.Rest_ExtEnable )
   END_RUNG
   RUNG wire#powerrail
      Contact( #AreaInterface.Man )
      I_Contact( #CIn.Manager.Control_ON )
      Contact( #Sts.OP_Ax_CanMoveFreely )
   END_RUNG wire#w1
   RUNG wire#powerrail
      I_Contact( #Ctrl.Ax.OP_MoveToPos )
      wire#w2
      Contact( #COut.Ax_InWPos )
      Contact( #Ax.COut.Standstill )
      wire#w3
      Coil( #Bloccaggio.Cin.Work_ExtEnable )
   END_RUNG
   RUNG wire#powerrail
      Contact( #CIn.Manager.Bloccaggio.Work )
   END_RUNG wire#w2
   RUNG wire#powerrail
      Contact( #AreaInterface.Man )
      I_Contact( #CIn.Manager.Control_ON )
      Contact( #Sts.OP_Ax_CanMoveFreely )
   END_RUNG wire#w3
   // the same network as SCL:
   #Bloccaggio.Cin.Rest_ExtEnable := #Ctrl.Ax.OP_MoveToPos OR (#AreaInterface.Man AND NOT #CIn.Manager.Control_ON AND #Sts.OP_Ax_CanMoveFreely);
   #Bloccaggio.Cin.Work_ExtEnable := ((NOT #Ctrl.Ax.OP_MoveToPos OR #CIn.Manager.Bloccaggio.Work) AND #COut.Ax_InWPos AND #Ax.COut.Standstill) OR (#AreaInterface.Man AND NOT #CIn.Manager.Control_ON AND #Sts.OP_Ax_CanMoveFreely);
END_REGION

REGION Network 36: [Bloccaggio] - Warning manacanza condizioni esecuzione Operazione RIPOSO / LAVORO
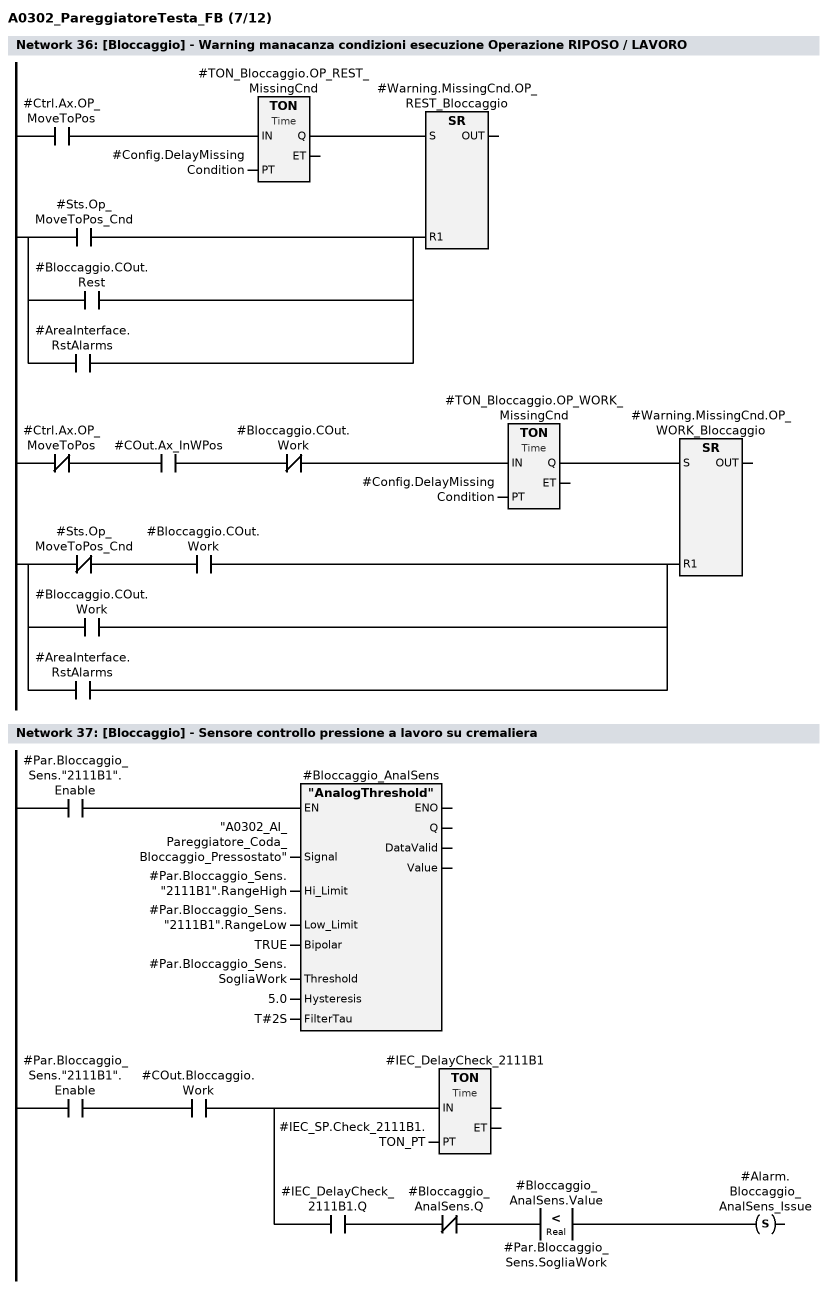
   RUNG wire#powerrail
      Contact( #Ctrl.Ax.OP_MoveToPos )
      { S7_Templates := "time_type := Time" } #TON_Bloccaggio.OP_REST_MissingCnd.TON(pt := #Config.DelayMissingCondition, et =>)
      S_SR(operand := #Warning.MissingCnd.OP_REST_Bloccaggio, r1 := wire#w1)
   END_RUNG
   RUNG wire#powerrail
      Contact( #Sts.Op_MoveToPos_Cnd )
   END_RUNG wire#w1
   RUNG wire#powerrail
      Contact( #Bloccaggio.COut.Rest )
   END_RUNG wire#w1
   RUNG wire#powerrail
      Contact( #AreaInterface.RstAlarms )
   END_RUNG wire#w1
   RUNG wire#powerrail
      I_Contact( #Ctrl.Ax.OP_MoveToPos )
      Contact( #COut.Ax_InWPos )
      I_Contact( #Bloccaggio.COut.Work )
      { S7_Templates := "time_type := Time" } #TON_Bloccaggio.OP_WORK_MissingCnd.TON(pt := #Config.DelayMissingCondition, et =>)
      S_SR(operand := #Warning.MissingCnd.OP_WORK_Bloccaggio, r1 := wire#w2)
   END_RUNG
   RUNG wire#powerrail
      I_Contact( #Sts.Op_MoveToPos_Cnd )
      Contact( #Bloccaggio.COut.Work )
   END_RUNG wire#w2
   RUNG wire#powerrail
      Contact( #Bloccaggio.COut.Work )
   END_RUNG wire#w2
   RUNG wire#powerrail
      Contact( #AreaInterface.RstAlarms )
   END_RUNG wire#w2
   // the same network as SCL:
   #TON_Bloccaggio.OP_REST_MissingCnd.TON(IN := #Ctrl.Ax.OP_MoveToPos, PT := #Config.DelayMissingCondition);
   IF #TON_Bloccaggio.OP_REST_MissingCnd.Q THEN
       #Warning.MissingCnd.OP_REST_Bloccaggio := TRUE;   // SR flip-flop
   END_IF;
   IF #Sts.Op_MoveToPos_Cnd OR #Bloccaggio.COut.Rest OR #AreaInterface.RstAlarms THEN
       #Warning.MissingCnd.OP_REST_Bloccaggio := FALSE;
   END_IF;
   #TON_Bloccaggio.OP_WORK_MissingCnd.TON(IN := NOT #Ctrl.Ax.OP_MoveToPos AND #COut.Ax_InWPos AND NOT #Bloccaggio.COut.Work,
                           PT := #Config.DelayMissingCondition);
   IF #TON_Bloccaggio.OP_WORK_MissingCnd.Q THEN
       #Warning.MissingCnd.OP_WORK_Bloccaggio := TRUE;   // SR flip-flop
   END_IF;
   IF (NOT #Sts.Op_MoveToPos_Cnd AND #Bloccaggio.COut.Work) OR #Bloccaggio.COut.Work OR #AreaInterface.RstAlarms THEN
       #Warning.MissingCnd.OP_WORK_Bloccaggio := FALSE;
   END_IF;
END_REGION

REGION Network 37: [Bloccaggio] - Sensore controllo pressione a lavoro su cremaliera
   RUNG wire#powerrail
      Contact( #Par.Bloccaggio_Sens."2111B1".Enable )
      #Bloccaggio_AnalSens(Signal := "A0302_AI_Pareggiatore_Coda_Bloccaggio_Pressostato", Hi_Limit := #Par.Bloccaggio_Sens."2111B1".RangeHigh, Low_Limit := #Par.Bloccaggio_Sens."2111B1".RangeLow, Bipolar := TRUE, Threshold := #Par.Bloccaggio_Sens.SogliaWork, Hysteresis := 5.0, FilterTau := T#2S, Q =>, DataValid =>, Value =>)
   END_RUNG
   RUNG wire#powerrail
      Contact( #Par.Bloccaggio_Sens."2111B1".Enable )
      Contact( #COut.Bloccaggio.Work )
      wire#w1
      { S7_Templates := "time_type := Time" } #IEC_DelayCheck_2111B1.TON(pt := #IEC_SP.Check_2111B1.TON_PT, et =>)
   END_RUNG
   RUNG wire#w1
      Contact( #IEC_DelayCheck_2111B1.Q )
      I_Contact( #Bloccaggio_AnalSens.Q )
      { S7_Templates := "SrcType := Real" } LT_Contact(in1 := #Bloccaggio_AnalSens.Value, in2 := #Par.Bloccaggio_Sens.SogliaWork)
      S_Coil( #Alarm.Bloccaggio_AnalSens_Issue )
   END_RUNG
   // the same network as SCL:
   IF #Par.Bloccaggio_Sens."2111B1".Enable THEN
       #Bloccaggio_AnalSens(Signal := "A0302_AI_Pareggiatore_Coda_Bloccaggio_Pressostato",   // "AnalogThreshold"
                            Hi_Limit := #Par.Bloccaggio_Sens."2111B1".RangeHigh,
                            Low_Limit := #Par.Bloccaggio_Sens."2111B1".RangeLow,
                            Bipolar := TRUE,
                            Threshold := #Par.Bloccaggio_Sens.SogliaWork,
                            Hysteresis := 5.0,
                            FilterTau := T#2S);
   END_IF;
   #_w1 := #Par.Bloccaggio_Sens."2111B1".Enable AND #COut.Bloccaggio.Work;
   #IEC_DelayCheck_2111B1.TON(IN := #_w1, PT := #IEC_SP.Check_2111B1.TON_PT);
   IF #_w1 AND #IEC_DelayCheck_2111B1.Q AND NOT #Bloccaggio_AnalSens.Q AND (#Bloccaggio_AnalSens.Value < #Par.Bloccaggio_Sens.SogliaWork) THEN
       #Alarm.Bloccaggio_AnalSens_Issue := TRUE;
   END_IF;
END_REGION

REGION Network 39 (SCL): == Calcolo setpoint posizione carri in funzione della cremaliera in Manuale ==
   // Foglio di calcolo posizione Cremaliera fornito
   // *****  Calcolo CARRO di TESTA ******

   IF #AreaInterface.Man AND #Ctrl.Ax.OP_MoveToPos THEN

       #CarroTesta.PosBattutePz := #Par.CarroPareggTesta.Preset;
       #CarroTesta.RimanenzaPos := (#Ax.HMI.TargetPosition - #CarroTesta.PosBattutePz);
       #CarroTesta.NrPassiReq := (#CarroTesta.RimanenzaPos / #Par.Cremaliera.Passo);

       // Calcolo i numeri di passi cremaliera richiesti per spostarmi della rimanenza
       #CarroTesta.PassoReq := ROUND(#CarroTesta.NrPassiReq);

       #Ax.Ctrl.Pos := (#CarroTesta.PassoReq * #Par.Cremaliera.Passo) + #CarroTesta.PosBattutePz;

   END_IF;
   (*
   IF #AreaInterface.Man AND #Ctrl.Ax.OP_MoveToPos THEN
       // Calcolo la rimanenza dello spazio tra lo 0 e il preset dei carri
       #CarroTesta.RimanenzaPos := #Ax.HMI.TargetPosition - #Par.CarroPareggTesta.Preset;

       // Calcolo i numeri di passi cremaliera richiesti per spostarmi della rimanenza
       #CarroTesta.PassoReq := ROUND(#CarroTesta.RimanenzaPos / #Par.Cremaliera.Passo);

       // Calcolo del setpoint di posizione dei 2 carri in funzione della misura calcolata - Se cambia il Beam Len viene richiesto il nuovo riposizionamento
       #Ax.Ctrl.Pos := (#CarroTesta.PassoReq * #Par.Cremaliera.Passo) + #Par.CarroPareggTesta.Preset;
   END_IF;
   *)
END_REGION

REGION Network 40: <<< AXIS >>>
END_REGION

REGION Network 41: [Ax] - CIn Dynamic Limits
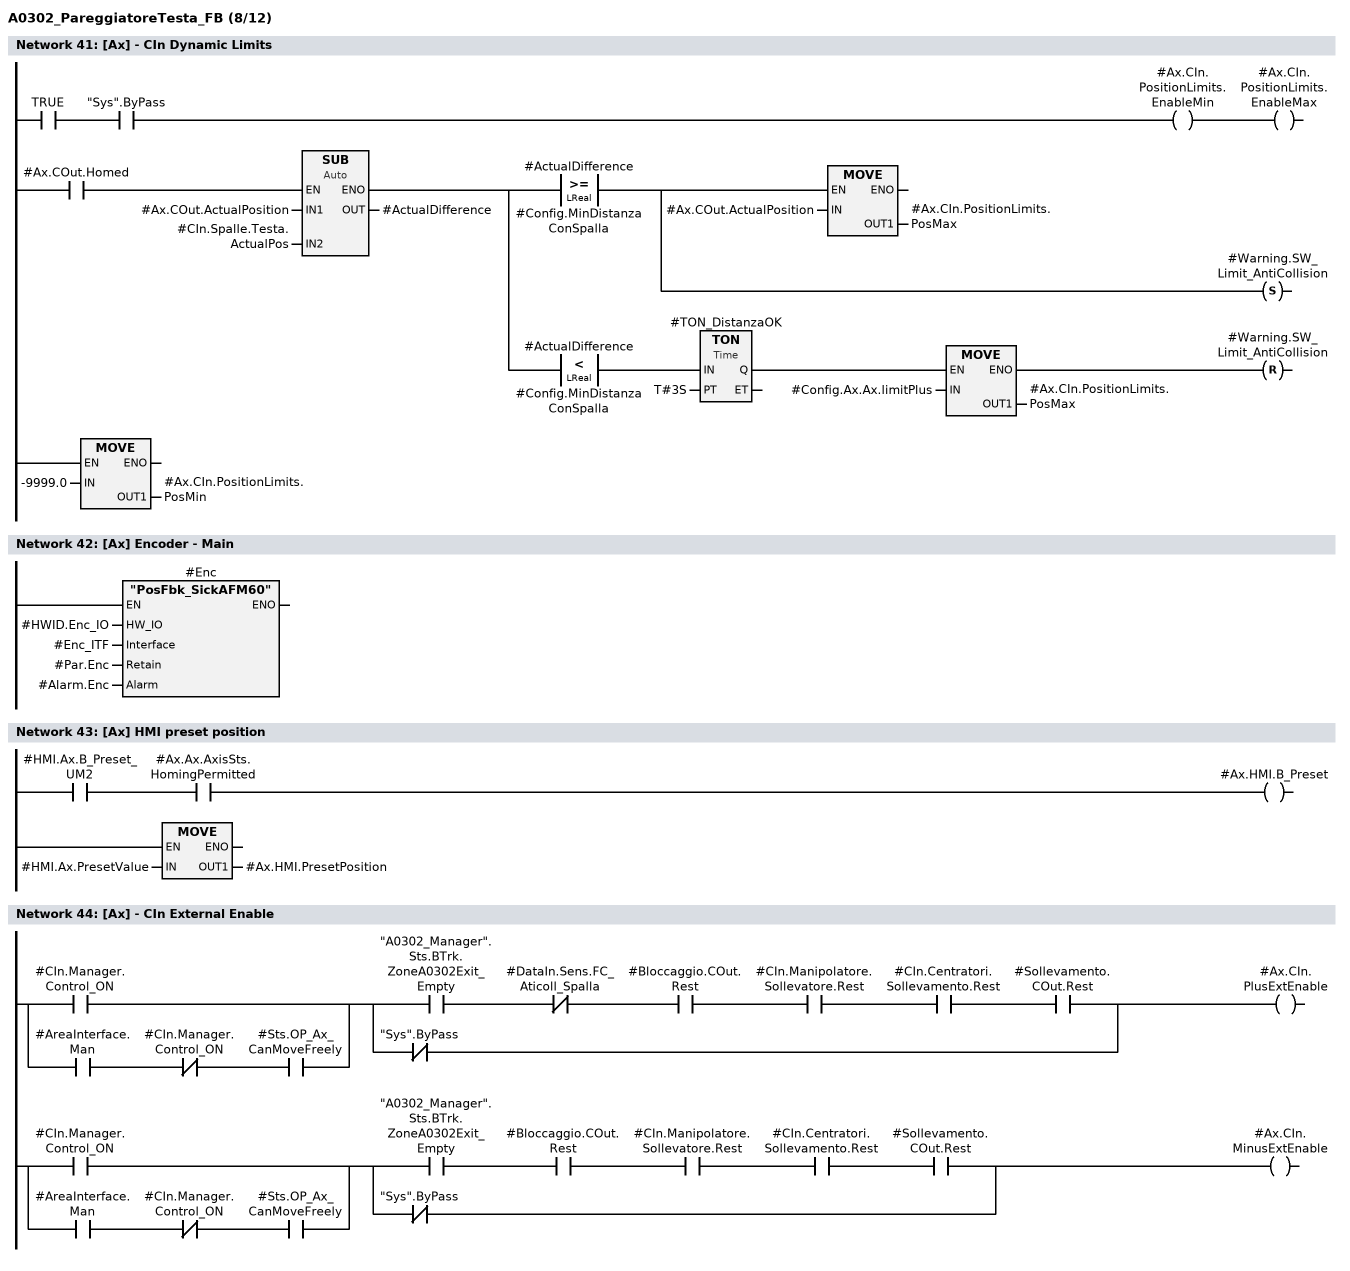
   RUNG wire#powerrail
      Contact( TRUE )
      Contact( "Sys".ByPass )
      Coil( #Ax.CIn.PositionLimits.EnableMin )
      Coil( #Ax.CIn.PositionLimits.EnableMax )
   END_RUNG
   RUNG wire#powerrail
      Contact( #Ax.COut.Homed )
      Sub(in1 := #Ax.COut.ActualPosition, in2 := #CIn.Spalle.Testa.ActualPos, out => #ActualDifference)
      wire#w1
      { S7_Templates := "SrcType := LReal" } GE_Contact(in1 := #ActualDifference, in2 := #Config.MinDistanzaConSpalla)
      wire#w2
      Move(in := #Ax.COut.ActualPosition, out1 => #Ax.CIn.PositionLimits.PosMax)
   END_RUNG
   RUNG wire#w2
      S_Coil( #Warning.SW_Limit_AntiCollision )
   END_RUNG
   RUNG wire#w1
      { S7_Templates := "SrcType := LReal" } LT_Contact(in1 := #ActualDifference, in2 := #Config.MinDistanzaConSpalla)
      { S7_Templates := "time_type := Time" } #TON_DistanzaOK.TON(pt := T#3S, et =>)
      Move(in := #Config.Ax.Ax.limitPlus, out1 => #Ax.CIn.PositionLimits.PosMax)
      R_Coil( #Warning.SW_Limit_AntiCollision )
   END_RUNG
   RUNG wire#powerrail
      Move(in := -9999.0, out1 => #Ax.CIn.PositionLimits.PosMin)
   END_RUNG
   // the same network as SCL:
   #Ax.CIn.PositionLimits.EnableMin := TRUE AND "Sys".ByPass;
   #Ax.CIn.PositionLimits.EnableMax := #Ax.CIn.PositionLimits.EnableMin;
   IF #Ax.COut.Homed THEN #ActualDifference := #Ax.COut.ActualPosition - #CIn.Spalle.Testa.ActualPos; END_IF;
   IF #Ax.COut.Homed AND (#ActualDifference >= #Config.MinDistanzaConSpalla) THEN
       #Ax.CIn.PositionLimits.PosMax := #Ax.COut.ActualPosition;
       #Warning.SW_Limit_AntiCollision := TRUE;
   END_IF;
   #TON_DistanzaOK.TON(IN := #Ax.COut.Homed AND (#ActualDifference < #Config.MinDistanzaConSpalla), PT := T#3S);
   IF #TON_DistanzaOK.Q THEN
       #Ax.CIn.PositionLimits.PosMax := #Config.Ax.Ax.limitPlus;
       #Warning.SW_Limit_AntiCollision := FALSE;
   END_IF;
   #Ax.CIn.PositionLimits.PosMin := -9999.0;
END_REGION

REGION Network 42: [Ax] Encoder - Main
   RUNG wire#powerrail
      #Enc(HW_IO := #HWID.Enc_IO, Interface := #Enc_ITF, Retain := #Par.Enc, Alarm := #Alarm.Enc)
   END_RUNG
   // the same network as SCL:
   #Enc(HW_IO := #HWID.Enc_IO, Interface := #Enc_ITF, Retain := #Par.Enc, Alarm := #Alarm.Enc);   // "PosFbk_SickAFM60"
END_REGION

REGION Network 43: [Ax] HMI preset position
   RUNG wire#powerrail
      Contact( #HMI.Ax.B_Preset_UM2 )
      Contact( #Ax.Ax.AxisSts.HomingPermitted )
      Coil( #Ax.HMI.B_Preset )
   END_RUNG
   RUNG wire#powerrail
      Move(in := #HMI.Ax.PresetValue, out1 => #Ax.HMI.PresetPosition)
   END_RUNG
   // the same network as SCL:
   #Ax.HMI.B_Preset := #HMI.Ax.B_Preset_UM2 AND #Ax.Ax.AxisSts.HomingPermitted;
   #Ax.HMI.PresetPosition := #HMI.Ax.PresetValue;
END_REGION

REGION Network 44: [Ax] - CIn External Enable
   RUNG wire#powerrail
      Contact( #CIn.Manager.Control_ON )
      wire#w1
      Contact( "A0302_Manager".Sts.BTrk.ZoneA0302Exit_Empty )
      I_Contact( #DataIn.Sens.FC_Aticoll_Spalla )
      Contact( #Bloccaggio.COut.Rest )
      Contact( #CIn.Manipolatore.Sollevatore.Rest )
      Contact( #CIn.Centratori.Sollevamento.Rest )
      Contact( #Sollevamento.COut.Rest )
      wire#w2
      Coil( #Ax.CIn.PlusExtEnable )
   END_RUNG
   RUNG wire#powerrail
      Contact( #AreaInterface.Man )
      I_Contact( #CIn.Manager.Control_ON )
      Contact( #Sts.OP_Ax_CanMoveFreely )
   END_RUNG wire#w1
   RUNG wire#w1
      I_Contact( "Sys".ByPass )
   END_RUNG wire#w2
   RUNG wire#powerrail
      Contact( #CIn.Manager.Control_ON )
      wire#w3
      Contact( "A0302_Manager".Sts.BTrk.ZoneA0302Exit_Empty )
      Contact( #Bloccaggio.COut.Rest )
      Contact( #CIn.Manipolatore.Sollevatore.Rest )
      Contact( #CIn.Centratori.Sollevamento.Rest )
      Contact( #Sollevamento.COut.Rest )
      wire#w4
      Coil( #Ax.CIn.MinusExtEnable )
   END_RUNG
   RUNG wire#powerrail
      Contact( #AreaInterface.Man )
      I_Contact( #CIn.Manager.Control_ON )
      Contact( #Sts.OP_Ax_CanMoveFreely )
   END_RUNG wire#w3
   RUNG wire#w3
      I_Contact( "Sys".ByPass )
   END_RUNG wire#w4
   // the same network as SCL:
   #Ax.CIn.PlusExtEnable := (#CIn.Manager.Control_ON OR (#AreaInterface.Man AND NOT #CIn.Manager.Control_ON AND #Sts.OP_Ax_CanMoveFreely)) AND (("A0302_Manager".Sts.BTrk.ZoneA0302Exit_Empty AND NOT #DataIn.Sens.FC_Aticoll_Spalla AND #Bloccaggio.COut.Rest AND #CIn.Manipolatore.Sollevatore.Rest AND #CIn.Centratori.Sollevamento.Rest AND #Sollevamento.COut.Rest) OR NOT "Sys".ByPass);
   #Ax.CIn.MinusExtEnable := (#CIn.Manager.Control_ON OR (#AreaInterface.Man AND NOT #CIn.Manager.Control_ON AND #Sts.OP_Ax_CanMoveFreely)) AND (("A0302_Manager".Sts.BTrk.ZoneA0302Exit_Empty AND #Bloccaggio.COut.Rest AND #CIn.Manipolatore.Sollevatore.Rest AND #CIn.Centratori.Sollevamento.Rest AND #Sollevamento.COut.Rest) OR NOT "Sys".ByPass);
END_REGION

REGION Network 45: [Ax] Axis Manager
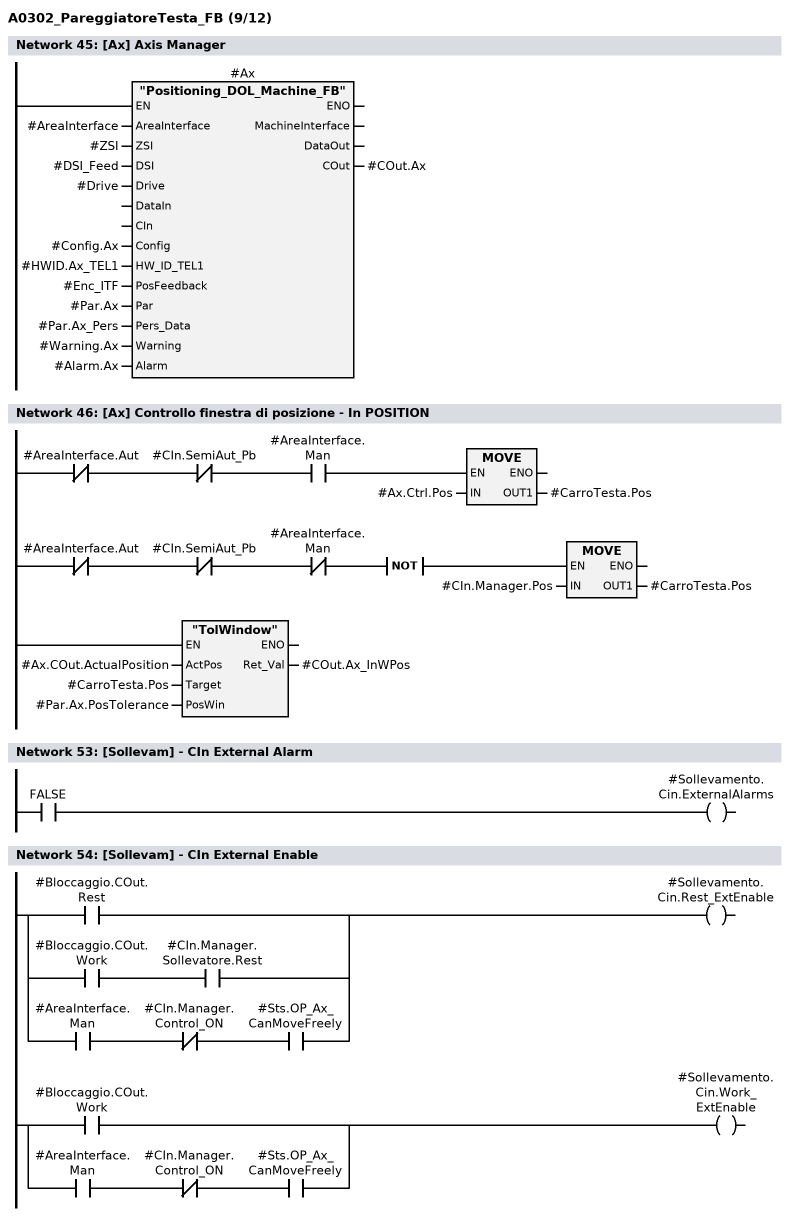
   RUNG wire#powerrail
      #Ax(AreaInterface := #AreaInterface, ZSI := #ZSI, DSI := #DSI_Feed, Drive := #Drive, DataIn :=, CIn :=, Config := #Config.Ax, HW_ID_TEL1 := #HWID.Ax_TEL1, PosFeedback := #Enc_ITF, Par := #Par.Ax, Pers_Data := #Par.Ax_Pers, Warning := #Warning.Ax, Alarm := #Alarm.Ax, MachineInterface =>, DataOut =>, COut => #COut.Ax)
   END_RUNG
   // the same network as SCL:
   #Ax(AreaInterface := #AreaInterface,   // "Positioning_DOL_Machine_FB"
       ZSI := #ZSI,
       DSI := #DSI_Feed,
       Drive := #Drive,
       Config := #Config.Ax,
       HW_ID_TEL1 := #HWID.Ax_TEL1,
       PosFeedback := #Enc_ITF,
       Par := #Par.Ax,
       Pers_Data := #Par.Ax_Pers,
       Warning := #Warning.Ax,
       Alarm := #Alarm.Ax,
       COut => #COut.Ax);
END_REGION

REGION Network 46: [Ax] Controllo finestra di posizione - In POSITION
   RUNG wire#powerrail
      I_Contact( #AreaInterface.Aut )
      I_Contact( #CIn.SemiAut_Pb )
      Contact( #AreaInterface.Man )
      Move(in := #Ax.Ctrl.Pos, out1 => #CarroTesta.Pos)
   END_RUNG
   RUNG wire#powerrail
      I_Contact( #AreaInterface.Aut )
      I_Contact( #CIn.SemiAut_Pb )
      I_Contact( #AreaInterface.Man )
      Not()
      Move(in := #CIn.Manager.Pos, out1 => #CarroTesta.Pos)
   END_RUNG
   RUNG wire#powerrail
      "TolWindow"(ActPos := #Ax.COut.ActualPosition, Target := #CarroTesta.Pos, PosWin := #Par.Ax.PosTolerance, Ret_Val => #COut.Ax_InWPos)
   END_RUNG
   // the same network as SCL:
   IF NOT #AreaInterface.Aut AND NOT #CIn.SemiAut_Pb AND #AreaInterface.Man THEN
       #CarroTesta.Pos := #Ax.Ctrl.Pos;
   END_IF;
   IF NOT (NOT #AreaInterface.Aut AND NOT #CIn.SemiAut_Pb AND NOT #AreaInterface.Man) THEN
       #CarroTesta.Pos := #CIn.Manager.Pos;
   END_IF;
   #COut.Ax_InWPos := "TolWindow"(ActPos := #Ax.COut.ActualPosition,
                           Target := #CarroTesta.Pos,
                           PosWin := #Par.Ax.PosTolerance);
END_REGION

REGION Network 47 (SCL): [Ax] - Cin Manager (Esecuzione sequenza comandi)
   // Operazione LAVORO dell' asse spintore quando i 2 ciclindri sono in riposo e il bloccaggio è a riposo
   #Ax.CIn.Manager.Control_ON := #Ax.DSI.PowerEnable := #Bloccaggio.Cin.Manager.Control_ON  := #Ctrl.Ax.OP_MoveToPos_Aut AND NOT #DataIn.Sens.FC_Aticoll_Spalla;

   IF #Ctrl.Ax.OP_MoveToPos_Aut AND #Sts.Op_MoveToPos_Cnd AND NOT #COut.Ax_InWPos AND #Bloccaggio.COut.Rest
           AND #Sollevamento.Cin.Manager.Rest AND #Centraggio.Cin.Manager.Rest THEN
           #Ax.CIn.Manager.MoveToPos := TRUE;

           // Se raggiungo la posizione di setpoint spengo il comando
       ELSIF #COut.Ax_InWPos AND #Ax.COut.Standstill THEN
           #Ax.CIn.Manager.MoveToPos := FALSE;
           #Ax.DSI.PowerEnable := FALSE;
       END_IF;

       // Attivazione ALLARME collisione con spalla
       // 
       IF #Ax.CIn.Manager.Control_ON AND #Ax.CIn.Manager.MoveToPos AND #DataIn.Sens.FC_Aticoll_Spalla THEN

           #Alarm.SensFC_Aticoll_Spalla := TRUE;
           #Ax.CIn.Manager.MoveToPos := FALSE;
           #Ax.DSI.PowerEnable := FALSE;
       END_IF;
END_REGION

REGION Network 48: <+>
END_REGION

REGION Network 49 (SCL): [Sollevam] - Cin Manager (Esecuzione sequenza comandi)
   // Comando CIn Manager ControlON di tutte le utenze
   #Sollevamento.Cin.Manager.Control_ON := (#Ctrl.Sollevamento.OP_Rest OR #Ctrl.Sollevamento.OP_Work) OR (#Ctrl.Centraggio.OP_Rest OR #Ctrl.Centraggio.OP_Work);

   #Sollevamento.Cin.Manager.Rest := FALSE;
   #Sollevamento.Cin.Manager.Work := FALSE;

   // Gestione dei comandi relativi a Battuta VRT in sequenza quando ho un OP cnd

   IF (#Ctrl.Sollevamento.OP_Rest AND #Sts.Sollevamento.OP_Rest_Cnd) OR (#Ctrl.Ax.OP_MoveToPos AND #Sts.Op_MoveToPos_Cnd) THEN

       #Sollevamento.Cin.Manager.Rest := #Centraggio.COut.Rest;

           // Vado a lavoro solo se sono in posizione e il carro è bloccato sulla cremaliera e i pezzi sono centrati sulla rulliera     
   ELSIF  (#Ctrl.Sollevamento.OP_Work AND #Sts.Sollevamento.Op_Work_Cnd) AND #Bloccaggio.COut.Work THEN

       #Sollevamento.Cin.Manager.Work := TRUE;
       #Centraggio.Cin.Manager.Rest := NOT #Sollevamento.COut.Work;

   END_IF;
END_REGION

REGION Network 50 (SCL): [Centraggio] - Cin Manager (Esecuzione sequenza comandi)
   // Comando CIn Manager ControlON di tutte le utenze
   #Centraggio.Cin.Manager.Control_ON := (#Ctrl.Centraggio.OP_Rest OR #Ctrl.Centraggio.OP_Work) OR (#Ctrl.Sollevamento.OP_Rest OR #Ctrl.Sollevamento.OP_Work);

   #Centraggio.Cin.Manager.Rest := FALSE;
   #Centraggio.Cin.Manager.Work := FALSE;

   // Gestione dei comandi relativi a Pareggiatore Longitudinale in sequenza quando ho un OP cnd
   IF (#Ctrl.Centraggio.OP_Rest AND #Sts.Centraggio.OP_Rest_Cnd) OR (#Ctrl.Ax.OP_MoveToPos AND #Sts.Op_MoveToPos_Cnd) THEN

       #Centraggio.Cin.Manager.Rest := TRUE;

           // Vado a lavoro solo se sono in posizione e il carro è bloccato sulla cremaliera e i pezzi sono centrati sulla rulliera     
   ELSIF  (#Ctrl.Centraggio.OP_Work AND #Sts.Centraggio.Op_Work_Cnd) AND #Bloccaggio.COut.Work THEN

       #Sollevamento.Cin.Manager.Work := TRUE;
       #Centraggio.Cin.Manager.Work := #Sollevamento.COut.Work;

   END_IF;
END_REGION

REGION Network 51: <+>
END_REGION

REGION Network 52: <<< SOLLEVAMENTO >>>
END_REGION

REGION Network 53: [Sollevam] - CIn External Alarm
   RUNG wire#powerrail
      Contact( FALSE )
      Coil( #Sollevamento.Cin.ExternalAlarms )
   END_RUNG
   // the same network as SCL:
   #Sollevamento.Cin.ExternalAlarms := FALSE;
END_REGION

REGION Network 54: [Sollevam] - CIn External Enable
   RUNG wire#powerrail
      Contact( #Bloccaggio.COut.Rest )
      wire#w1
      Coil( #Sollevamento.Cin.Rest_ExtEnable )
   END_RUNG
   RUNG wire#powerrail
      Contact( #Bloccaggio.COut.Work )
      Contact( #CIn.Manager.Sollevatore.Rest )
   END_RUNG wire#w1
   RUNG wire#powerrail
      Contact( #AreaInterface.Man )
      I_Contact( #CIn.Manager.Control_ON )
      Contact( #Sts.OP_Ax_CanMoveFreely )
   END_RUNG wire#w1
   RUNG wire#powerrail
      Contact( #Bloccaggio.COut.Work )
      wire#w2
      Coil( #Sollevamento.Cin.Work_ExtEnable )
   END_RUNG
   RUNG wire#powerrail
      Contact( #AreaInterface.Man )
      I_Contact( #CIn.Manager.Control_ON )
      Contact( #Sts.OP_Ax_CanMoveFreely )
   END_RUNG wire#w2
   // the same network as SCL:
   #Sollevamento.Cin.Rest_ExtEnable := #Bloccaggio.COut.Rest OR (#Bloccaggio.COut.Work AND #CIn.Manager.Sollevatore.Rest) OR (#AreaInterface.Man AND NOT #CIn.Manager.Control_ON AND #Sts.OP_Ax_CanMoveFreely);
   #Sollevamento.Cin.Work_ExtEnable := #Bloccaggio.COut.Work OR (#AreaInterface.Man AND NOT #CIn.Manager.Control_ON AND #Sts.OP_Ax_CanMoveFreely);
END_REGION

REGION Network 55: [Sollevam] - Warning manacanza condizioni esecuzione Operazione RIPOSO / LAVORO
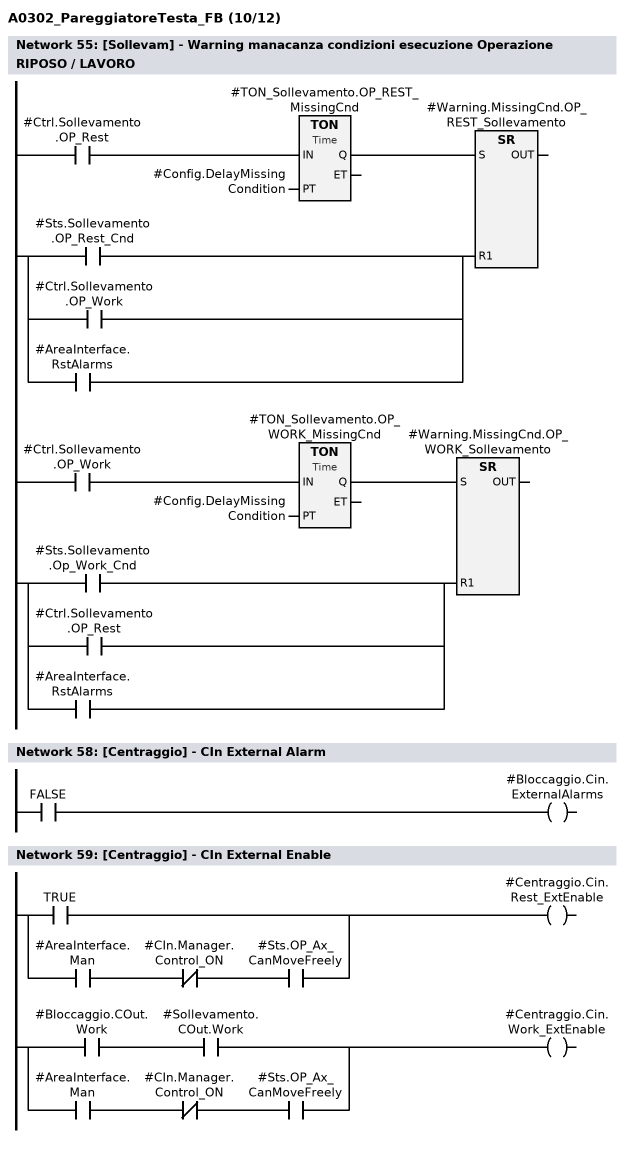
   RUNG wire#powerrail
      Contact( #Ctrl.Sollevamento.OP_Rest )
      { S7_Templates := "time_type := Time" } #TON_Sollevamento.OP_REST_MissingCnd.TON(pt := #Config.DelayMissingCondition, et =>)
      S_SR(operand := #Warning.MissingCnd.OP_REST_Sollevamento, r1 := wire#w1)
   END_RUNG
   RUNG wire#powerrail
      Contact( #Sts.Sollevamento.OP_Rest_Cnd )
   END_RUNG wire#w1
   RUNG wire#powerrail
      Contact( #Ctrl.Sollevamento.OP_Work )
   END_RUNG wire#w1
   RUNG wire#powerrail
      Contact( #AreaInterface.RstAlarms )
   END_RUNG wire#w1
   RUNG wire#powerrail
      Contact( #Ctrl.Sollevamento.OP_Work )
      { S7_Templates := "time_type := Time" } #TON_Sollevamento.OP_WORK_MissingCnd.TON(pt := #Config.DelayMissingCondition, et =>)
      S_SR(operand := #Warning.MissingCnd.OP_WORK_Sollevamento, r1 := wire#w2)
   END_RUNG
   RUNG wire#powerrail
      Contact( #Sts.Sollevamento.Op_Work_Cnd )
   END_RUNG wire#w2
   RUNG wire#powerrail
      Contact( #Ctrl.Sollevamento.OP_Rest )
   END_RUNG wire#w2
   RUNG wire#powerrail
      Contact( #AreaInterface.RstAlarms )
   END_RUNG wire#w2
   // the same network as SCL:
   #TON_Sollevamento.OP_REST_MissingCnd.TON(IN := #Ctrl.Sollevamento.OP_Rest,
                           PT := #Config.DelayMissingCondition);
   IF #TON_Sollevamento.OP_REST_MissingCnd.Q THEN
       #Warning.MissingCnd.OP_REST_Sollevamento := TRUE;   // SR flip-flop
   END_IF;
   IF #Sts.Sollevamento.OP_Rest_Cnd OR #Ctrl.Sollevamento.OP_Work OR #AreaInterface.RstAlarms THEN
       #Warning.MissingCnd.OP_REST_Sollevamento := FALSE;
   END_IF;
   #TON_Sollevamento.OP_WORK_MissingCnd.TON(IN := #Ctrl.Sollevamento.OP_Work,
                           PT := #Config.DelayMissingCondition);
   IF #TON_Sollevamento.OP_WORK_MissingCnd.Q THEN
       #Warning.MissingCnd.OP_WORK_Sollevamento := TRUE;   // SR flip-flop
   END_IF;
   IF #Sts.Sollevamento.Op_Work_Cnd OR #Ctrl.Sollevamento.OP_Rest OR #AreaInterface.RstAlarms THEN
       #Warning.MissingCnd.OP_WORK_Sollevamento := FALSE;
   END_IF;
END_REGION

REGION Network 57: <<< CENTRAGGIO >>>
END_REGION

REGION Network 58: [Centraggio] - CIn External Alarm
   RUNG wire#powerrail
      Contact( FALSE )
      Coil( #Bloccaggio.Cin.ExternalAlarms )
   END_RUNG
   // the same network as SCL:
   #Bloccaggio.Cin.ExternalAlarms := FALSE;
END_REGION

REGION Network 59: [Centraggio] - CIn External Enable
   RUNG wire#powerrail
      Contact( TRUE )
      wire#w1
      Coil( #Centraggio.Cin.Rest_ExtEnable )
   END_RUNG
   RUNG wire#powerrail
      Contact( #AreaInterface.Man )
      I_Contact( #CIn.Manager.Control_ON )
      Contact( #Sts.OP_Ax_CanMoveFreely )
   END_RUNG wire#w1
   RUNG wire#powerrail
      Contact( #Bloccaggio.COut.Work )
      Contact( #Sollevamento.COut.Work )
      wire#w2
      Coil( #Centraggio.Cin.Work_ExtEnable )
   END_RUNG
   RUNG wire#powerrail
      Contact( #AreaInterface.Man )
      I_Contact( #CIn.Manager.Control_ON )
      Contact( #Sts.OP_Ax_CanMoveFreely )
   END_RUNG wire#w2
   // the same network as SCL:
   #Centraggio.Cin.Rest_ExtEnable := TRUE OR (#AreaInterface.Man AND NOT #CIn.Manager.Control_ON AND #Sts.OP_Ax_CanMoveFreely);
   #Centraggio.Cin.Work_ExtEnable := (#Bloccaggio.COut.Work AND #Sollevamento.COut.Work) OR (#AreaInterface.Man AND NOT #CIn.Manager.Control_ON AND #Sts.OP_Ax_CanMoveFreely);
END_REGION

REGION Network 60: [Centraggio] - Warning manacanza condizioni esecuzione Operazione RIPOSO / LAVORO
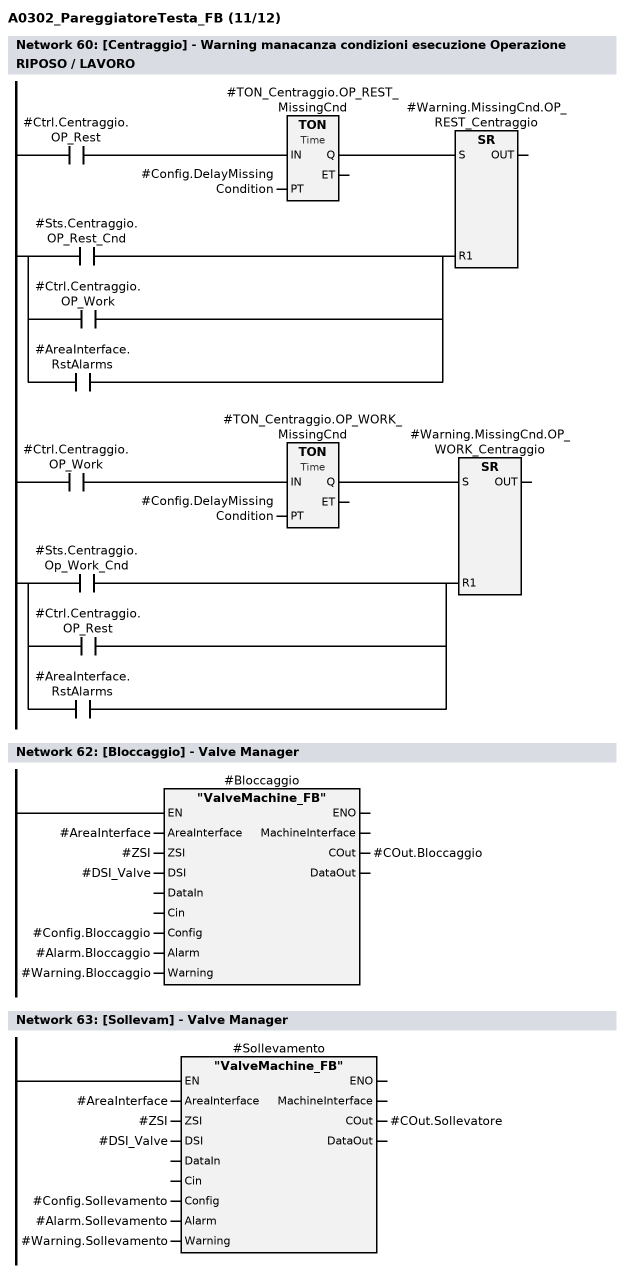
   RUNG wire#powerrail
      Contact( #Ctrl.Centraggio.OP_Rest )
      { S7_Templates := "time_type := Time" } #TON_Centraggio.OP_REST_MissingCnd.TON(pt := #Config.DelayMissingCondition, et =>)
      S_SR(operand := #Warning.MissingCnd.OP_REST_Centraggio, r1 := wire#w1)
   END_RUNG
   RUNG wire#powerrail
      Contact( #Sts.Centraggio.OP_Rest_Cnd )
   END_RUNG wire#w1
   RUNG wire#powerrail
      Contact( #Ctrl.Centraggio.OP_Work )
   END_RUNG wire#w1
   RUNG wire#powerrail
      Contact( #AreaInterface.RstAlarms )
   END_RUNG wire#w1
   RUNG wire#powerrail
      Contact( #Ctrl.Centraggio.OP_Work )
      { S7_Templates := "time_type := Time" } #TON_Centraggio.OP_WORK_MissingCnd.TON(pt := #Config.DelayMissingCondition, et =>)
      S_SR(operand := #Warning.MissingCnd.OP_WORK_Centraggio, r1 := wire#w2)
   END_RUNG
   RUNG wire#powerrail
      Contact( #Sts.Centraggio.Op_Work_Cnd )
   END_RUNG wire#w2
   RUNG wire#powerrail
      Contact( #Ctrl.Centraggio.OP_Rest )
   END_RUNG wire#w2
   RUNG wire#powerrail
      Contact( #AreaInterface.RstAlarms )
   END_RUNG wire#w2
   // the same network as SCL:
   #TON_Centraggio.OP_REST_MissingCnd.TON(IN := #Ctrl.Centraggio.OP_Rest, PT := #Config.DelayMissingCondition);
   IF #TON_Centraggio.OP_REST_MissingCnd.Q THEN
       #Warning.MissingCnd.OP_REST_Centraggio := TRUE;   // SR flip-flop
   END_IF;
   IF #Sts.Centraggio.OP_Rest_Cnd OR #Ctrl.Centraggio.OP_Work OR #AreaInterface.RstAlarms THEN
       #Warning.MissingCnd.OP_REST_Centraggio := FALSE;
   END_IF;
   #TON_Centraggio.OP_WORK_MissingCnd.TON(IN := #Ctrl.Centraggio.OP_Work, PT := #Config.DelayMissingCondition);
   IF #TON_Centraggio.OP_WORK_MissingCnd.Q THEN
       #Warning.MissingCnd.OP_WORK_Centraggio := TRUE;   // SR flip-flop
   END_IF;
   IF #Sts.Centraggio.Op_Work_Cnd OR #Ctrl.Centraggio.OP_Rest OR #AreaInterface.RstAlarms THEN
       #Warning.MissingCnd.OP_WORK_Centraggio := FALSE;
   END_IF;
END_REGION

REGION Network 62: [Bloccaggio] - Valve Manager
   RUNG wire#powerrail
      #Bloccaggio(AreaInterface := #AreaInterface, ZSI := #ZSI, DSI := #DSI_Valve, DataIn :=, Cin :=, Config := #Config.Bloccaggio, Alarm := #Alarm.Bloccaggio, Warning := #Warning.Bloccaggio, MachineInterface =>, COut => #COut.Bloccaggio, DataOut =>)
   END_RUNG
   // the same network as SCL:
   #Bloccaggio(AreaInterface := #AreaInterface,   // "ValveMachine_FB"
               ZSI := #ZSI,
               DSI := #DSI_Valve,
               Config := #Config.Bloccaggio,
               Alarm := #Alarm.Bloccaggio,
               Warning := #Warning.Bloccaggio,
               COut => #COut.Bloccaggio);
END_REGION

REGION Network 63: [Sollevam] - Valve Manager
   RUNG wire#powerrail
      #Sollevamento(AreaInterface := #AreaInterface, ZSI := #ZSI, DSI := #DSI_Valve, DataIn :=, Cin :=, Config := #Config.Sollevamento, Alarm := #Alarm.Sollevamento, Warning := #Warning.Sollevamento, MachineInterface =>, COut => #COut.Sollevatore, DataOut =>)
   END_RUNG
   // the same network as SCL:
   #Sollevamento(AreaInterface := #AreaInterface,   // "ValveMachine_FB"
                 ZSI := #ZSI,
                 DSI := #DSI_Valve,
                 Config := #Config.Sollevamento,
                 Alarm := #Alarm.Sollevamento,
                 Warning := #Warning.Sollevamento,
                 COut => #COut.Sollevatore);
END_REGION

REGION Network 64 (SCL): [Sollevam] - Anticipo COut
   #COut.Sollevatore := #Sollevamento.COut;

   #COut.Sollevatore.Rest := #Sollevamento.COut.Rest OR #TON_Anticipi.Rest.Sollevamento.Q;
   #COut.Sollevatore.Work := #Sollevamento.COut.Work OR #TON_Anticipi.Work.Sollevamento.Q;
END_REGION

REGION Network 65: [Centraggio] - Valve Manager
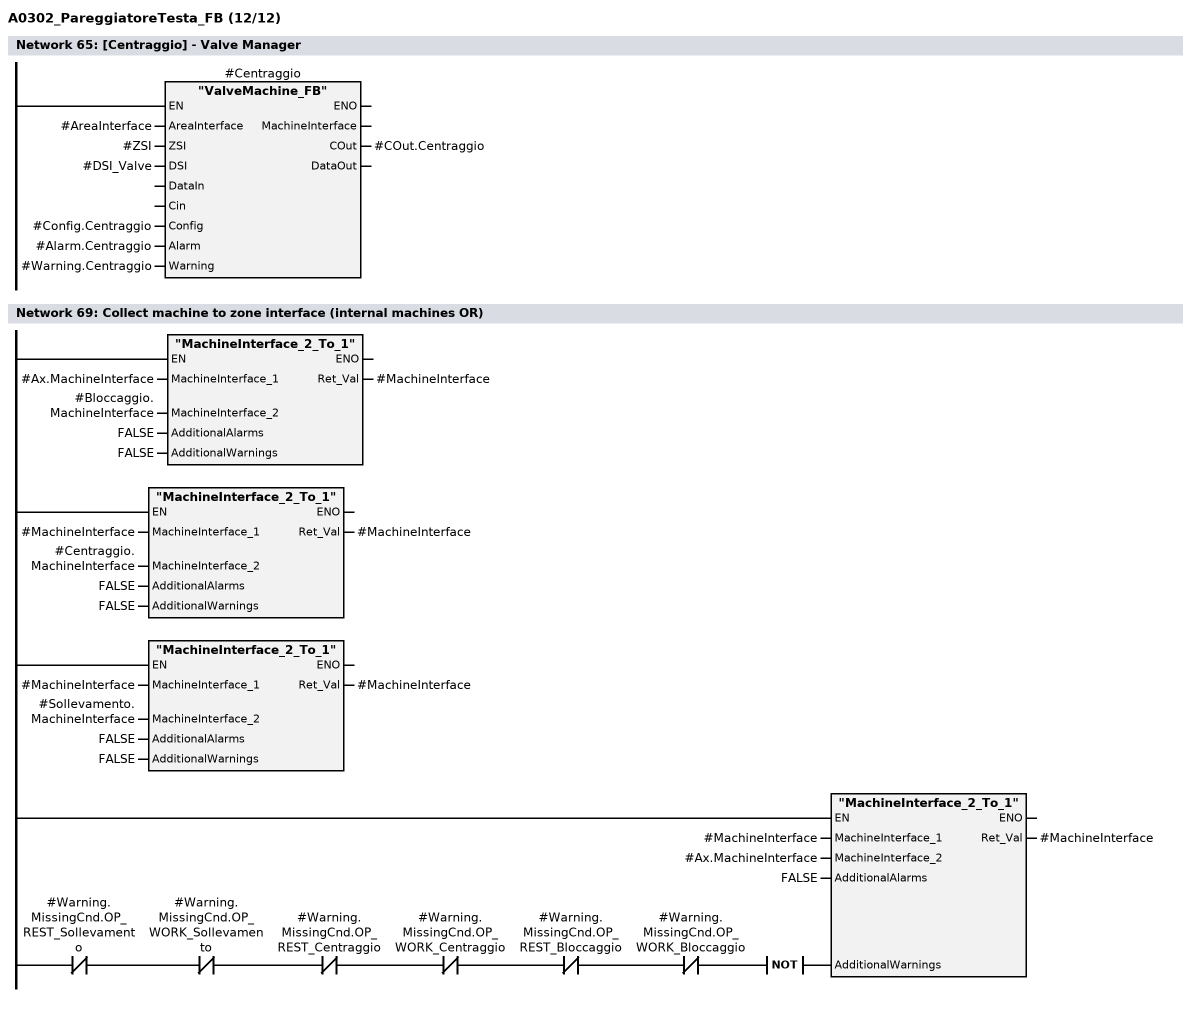
   RUNG wire#powerrail
      #Centraggio(AreaInterface := #AreaInterface, ZSI := #ZSI, DSI := #DSI_Valve, DataIn :=, Cin :=, Config := #Config.Centraggio, Alarm := #Alarm.Centraggio, Warning := #Warning.Centraggio, MachineInterface =>, COut => #COut.Centraggio, DataOut =>)
   END_RUNG
   // the same network as SCL:
   #Centraggio(AreaInterface := #AreaInterface,   // "ValveMachine_FB"
               ZSI := #ZSI,
               DSI := #DSI_Valve,
               Config := #Config.Centraggio,
               Alarm := #Alarm.Centraggio,
               Warning := #Warning.Centraggio,
               COut => #COut.Centraggio);
END_REGION

REGION Network 66 (SCL): [Centraggio] - Anticipo COut
   #COut.Centraggio := #Centraggio.COut;

   #COut.Centraggio.Rest := #Centraggio.COut.Rest OR #TON_Anticipi.Rest.Centraggio.Q;
   #COut.Centraggio.Work:= #Centraggio.COut.Work OR #TON_Anticipi.Work.Centraggio.Q;
END_REGION

REGION Network 68: <<< MACHINE STATUS >>>
END_REGION

REGION Network 69: Collect machine to zone interface (internal machines OR)
   RUNG wire#powerrail
      "MachineInterface_2_To_1"(MachineInterface_1 := #Ax.MachineInterface, MachineInterface_2 := #Bloccaggio.MachineInterface, AdditionalAlarms := FALSE, AdditionalWarnings := FALSE, Ret_Val => #MachineInterface)
   END_RUNG
   RUNG wire#powerrail
      "MachineInterface_2_To_1"(MachineInterface_1 := #MachineInterface, MachineInterface_2 := #Centraggio.MachineInterface, AdditionalAlarms := FALSE, AdditionalWarnings := FALSE, Ret_Val => #MachineInterface)
   END_RUNG
   RUNG wire#powerrail
      "MachineInterface_2_To_1"(MachineInterface_1 := #MachineInterface, MachineInterface_2 := #Sollevamento.MachineInterface, AdditionalAlarms := FALSE, AdditionalWarnings := FALSE, Ret_Val => #MachineInterface)
   END_RUNG
   RUNG wire#powerrail
      "MachineInterface_2_To_1"(AdditionalWarnings := wire#w1, MachineInterface_1 := #MachineInterface, MachineInterface_2 := #Ax.MachineInterface, AdditionalAlarms := FALSE, Ret_Val => #MachineInterface)
   END_RUNG
   RUNG wire#powerrail
      I_Contact( #Warning.MissingCnd.OP_REST_Sollevamento )
      I_Contact( #Warning.MissingCnd.OP_WORK_Sollevamento )
      I_Contact( #Warning.MissingCnd.OP_REST_Centraggio )
      I_Contact( #Warning.MissingCnd.OP_WORK_Centraggio )
      I_Contact( #Warning.MissingCnd.OP_REST_Bloccaggio )
      I_Contact( #Warning.MissingCnd.OP_WORK_Bloccaggio )
      Not()
   END_RUNG wire#w1
   // the same network as SCL:
   #MachineInterface := "MachineInterface_2_To_1"(MachineInterface_1 := #Ax.MachineInterface,
                           MachineInterface_2 := #Bloccaggio.MachineInterface,
                           AdditionalAlarms := FALSE,
                           AdditionalWarnings := FALSE);
   #MachineInterface := "MachineInterface_2_To_1"(MachineInterface_1 := #MachineInterface,
                           MachineInterface_2 := #Centraggio.MachineInterface,
                           AdditionalAlarms := FALSE,
                           AdditionalWarnings := FALSE);
   #MachineInterface := "MachineInterface_2_To_1"(MachineInterface_1 := #MachineInterface,
                           MachineInterface_2 := #Sollevamento.MachineInterface,
                           AdditionalAlarms := FALSE,
                           AdditionalWarnings := FALSE);
   #MachineInterface := "MachineInterface_2_To_1"(MachineInterface_1 := #MachineInterface,
                           MachineInterface_2 := #Ax.MachineInterface,
                           AdditionalAlarms := FALSE,
                           AdditionalWarnings := NOT (NOT #Warning.MissingCnd.OP_REST_Sollevamento AND NOT #Warning.MissingCnd.OP_WORK_Sollevamento AND NOT #Warning.MissingCnd.OP_REST_Centraggio AND NOT #Warning.MissingCnd.OP_WORK_Centraggio AND NOT #Warning.MissingCnd.OP_REST_Bloccaggio AND NOT #Warning.MissingCnd.OP_WORK_Bloccaggio));
END_REGION
END_FUNCTION_BLOCK
